T1906 BOOL  ; #1-1腔体氦检数据取值判定延时（测试）
T1907 BOOL  ; #1-1腔体抽残气压力到达延时（测试）
T1908 BOOL  ; #1-1腔体抽残气时间上限到达延时（测试）
T1909 BOOL  ; #1-1腔体预抽时间到达延时（测试）
T1910 BOOL  ; $?St$Bk?_#[195] / #1-1腔体真空在可氦检状态（测试） / $?St$Bk?_#[195]
T1920 BOOL  ; #1-1电池抽真空阈值到达延时（测试）
T1921 BOOL  ; #1-1电池抽真空时间上限到达延时（测试）
T1922 BOOL  ; #1-1电池破真空阈值到达延时（测试）
T1923 BOOL  ; #1-1电池破真空时间上限到达延时（测试）
T1924 BOOL  ; #1-1电池注氦压力到达延时（测试）
T1925 BOOL  ; #1-1电池注氦时间上限到达延时（测试）
T1926 BOOL  ; #1-1电池抽残气压力到达延时（测试）
T1927 BOOL  ; #1-1电池抽残气时间上限到达延时（测试）
T1928 BOOL  ; #1-1电池预抽压力正常判定延时（测试）
T1940 BOOL  ; 数据初始化延时（清氦）
T1941 BOOL  ; 清氦注氮时长（清氦）
T1980 BOOL  ; #1-1腔体数据初始化延时（标漏）
T1981 BOOL  ; #1-1腔体抽真空阀值到达延时（标漏）
T1982 BOOL  ; #1-1腔体抽真空时间上限到达延时（标漏）
T1984 BOOL  ; #1-1腔体氦检延时（标漏）
T1985 BOOL  ; #1-1腔体氦检数据取值完成判定（标漏）
T1986 BOOL  ; 氦检阀打开后，腔体压力超过氦检安全阀值，判氦检异常（标漏）
T1987 BOOL  ; 开氦检阀前抽气阀关延时（标漏）
T1990 BOOL  ; 氦检仪稳定延时（公共）
T2000 BOOL  ; #2-1腔体抽真空阈值到达延时（测试）
T2001 BOOL  ; #2-1腔体抽真空时间上限到达延时（测试）
T2002 BOOL  ; #2-1腔体破真空阈值到达延时（测试）
T2004 BOOL  ; #2-1腔体氦检时间（测试）
T2005 BOOL  ; #2-1腔体抽气阀关闭延时（测试）
T2006 BOOL  ; #2-1腔体氦检数据取值判定延时（测试）
T2007 BOOL  ; #2-1腔体抽残气压力到达延时（测试）
T2008 BOOL  ; #2-1腔体抽残气时间上限到达延时（测试）
T2009 BOOL  ; #2-1腔体预抽时间到达延时（测试）
T2010 BOOL  ; #2-1腔体真空在可氦检状态（测试）
T2020 BOOL  ; #2-1电池抽真空阈值到达延时（测试）
T2021 BOOL  ; #2-1电池抽真空时间上限到达延时（测试）
T2022 BOOL  ; #2-1电池破真空阈值到达延时（测试）
T2023 BOOL  ; #2-1电池破真空时间上限到达延时（测试）
T2024 BOOL  ; #2-1电池注氦压力到达延时（测试）
T2025 BOOL  ; #2-1电池注氦时间上限到达延时（测试）
T2026 BOOL  ; #2-1电池抽残气压力到达延时（测试）
T2027 BOOL  ; #2-1电池抽残气时间上限到达延时（测试）
T2028 BOOL  ; #2-1电池预抽压力正常判定延时（测试）
T2040 BOOL  ; #2-1数据初始化延时（清氦）
T2041 BOOL  ; #2-1清氦注氮时长（清氦）
T2081 BOOL  ; #2-1腔体抽真空阀值到达延时（标漏）
T2082 BOOL  ; #2-1腔体抽真空时间上限到达延时（标漏）
T2084 BOOL  ; #2-1腔体氦检延时（标漏）
T2085 BOOL  ; #2-1腔体氦检数据取值完成判定（标漏）
T2086 BOOL  ; #2-1氦检阀打开后，腔体压力超过氦检安全阀值，判氦检异常（标漏）
T2087 BOOL  ; #2-1开氦检阀前抽气阀关延时（标漏）
T2100 BOOL  ; #3-1腔体抽真空阈值到达延时（测试）
T2101 BOOL  ; #3-1腔体抽真空时间上限到达延时（测试）
T2102 BOOL  ; #3-1腔体破真空阈值到达延时（测试）
T2104 BOOL  ; #3-1腔体氦检时间（测试）
T2105 BOOL  ; #3-1腔体抽气阀关闭延时（测试）
T2106 BOOL  ; #3-1腔体氦检数据取值判定延时（测试）
T2107 BOOL  ; #3-1腔体抽残气压力到达延时（测试）
T2108 BOOL  ; #3-1腔体抽残气时间上限到达延时（测试）
T2109 BOOL  ; #3-1腔体预抽时间到达延时（测试）
T2110 BOOL  ; #3-1腔体真空在可氦检状态（测试）
T2120 BOOL  ; #3-1电池抽真空阈值到达延时（测试）
T2121 BOOL  ; #3-1电池抽真空时间上限到达延时（测试）
T2122 BOOL  ; #3-1电池破真空阈值到达延时（测试）
T2123 BOOL  ; #3-1电池破真空时间上限到达延时（测试）
T2124 BOOL  ; #3-1电池注氦压力到达延时（测试）
T2125 BOOL  ; #3-1电池注氦时间上限到达延时（测试）
T2126 BOOL  ; #3-1电池抽残气压力到达延时（测试）
T2127 BOOL  ; #3-1电池抽残气时间上限到达延时（测试）
T2128 BOOL  ; #3-1电池预抽压力正常判定延时（测试）
T2140 BOOL  ; #3-1数据初始化延时（清氦）
T2141 BOOL  ; #3-1清氦注氮时长（清氦）
T2181 BOOL  ; #3-1腔体抽真空阀值到达延时（标漏）
T2182 BOOL  ; #3-1腔体抽真空时间上限到达延时（标漏）
T2184 BOOL  ; #3-1腔体氦检延时（标漏）
T2185 BOOL  ; #3-1腔体氦检数据取值完成判定（标漏）
T2186 BOOL  ; #3-1氦检阀打开后，腔体压力超过氦检安全阀值，判氦检异常（标漏）
T2187 BOOL  ; #3-1开氦检阀前抽气阀关延时（标漏）
T2220 BOOL  ; #1-2电池抽真空阈值到达延时（测试）
T2221 BOOL  ; #1-2电池抽真空时间上限到达延时（测试）
T2222 BOOL  ; #1-2电池破真空阈值到达延时（测试）
T2223 BOOL  ; #1-2电池破真空时间上限到达延时（测试）
T2224 BOOL  ; #1-2电池注氦压力到达延时（测试）
T2225 BOOL  ; #1-2电池注氦时间上限到达延时（测试）
T2226 BOOL  ; #1-2电池抽残气压力到达延时（测试）
T2227 BOOL  ; #1-2电池抽残气时间上限到达延时（测试）
T2228 BOOL  ; #1-2电池预抽压力正常判定延时（测试）
T2281 BOOL  ; #1-2腔体抽真空阀值到达延时（标漏）
T2282 BOOL  ; #1-2腔体抽真空时间上限到达延时（标漏）
T2284 BOOL  ; #1-2腔体氦检延时（标漏）
T2286 BOOL  ; #1-2氦检阀打开后，腔体压力超过氦检安全阀值，判氦检异常（标漏）
T2287 BOOL  ; #1-2开氦检阀前抽气阀关延时（标漏）
T2320 BOOL  ; #2-2电池抽真空阈值到达延时（测试）
T2321 BOOL  ; #2-2电池抽真空时间上限到达延时（测试）
T2322 BOOL  ; #2-2电池破真空阈值到达延时（测试）
T2323 BOOL  ; #2-2电池破真空时间上限到达延时（测试）
T2324 BOOL  ; #2-2电池注氦压力到达延时（测试）
T2325 BOOL  ; #2-2电池注氦时间上限到达延时（测试）
T2326 BOOL  ; #2-2电池抽残气压力到达延时（测试）
T2327 BOOL  ; #2-2电池抽残气时间上限到达延时（测试）
T2328 BOOL  ; #2-2电池预抽压力正常判定延时（测试）
T2381 BOOL  ; #2-2腔体抽真空阀值到达延时（标漏）
T2382 BOOL  ; #2-2腔体抽真空时间上限到达延时（标漏）
T2384 BOOL  ; #2-2腔体氦检延时（标漏）
T2386 BOOL  ; #2-2氦检阀打开后，腔体压力超过氦检安全阀值，判氦检异常（标漏）
T2387 BOOL  ; #2-2开氦检阀前抽气阀关延时（标漏）
T2420 BOOL  ; #3-2电池抽真空阈值到达延时（测试）
T2421 BOOL  ; #3-2电池抽真空时间上限到达延时（测试）
T2422 BOOL  ; #3-2电池破真空阈值到达延时（测试）
T2423 BOOL  ; #3-2电池破真空时间上限到达延时（测试）
T2424 BOOL  ; #3-2电池注氦压力到达延时（测试）
T2425 BOOL  ; #3-2电池注氦时间上限到达延时（测试）
T2426 BOOL  ; #3-2电池抽残气压力到达延时（测试）
T2427 BOOL  ; #3-2电池抽残气时间上限到达延时（测试）
T2428 BOOL  ; #3-2电池预抽压力正常判定延时（测试）
T2481 BOOL  ; #3-2腔体抽真空阀值到达延时（标漏）
T2482 BOOL  ; #3-2腔体抽真空时间上限到达延时（标漏）
T2484 BOOL  ; #3-2腔体氦检延时（标漏）
T2486 BOOL  ; #3-2氦检阀打开后，腔体压力超过氦检安全阀值，判氦检异常（标漏）
T2487 BOOL  ; #3-2开氦检阀前抽气阀关延时（标漏）
T2521 BOOL  ; 进料#1扫码延时
T2522 BOOL  ; 接收数据清零延时发送无协议通讯TXD
T2523 BOOL  ; 进料#1扫码结果判定延时
T2524 BOOL  ; 进料#1扫码发送超时
T2531 BOOL  ; 进料#2扫码延时
T2532 BOOL  ; 扫码长度判定延时
T2600 BOOL  ; #4-1腔体抽真空阈值到达延时（测试）
T2601 BOOL  ; #4-1腔体抽真空时间上限到达延时（测试）
T2602 BOOL  ; #4-1腔体破真空阈值到达延时（测试）
T2603 BOOL  ; #4-1腔体破真空时间上限到达延时（测试）
T2604 BOOL  ; #4-1腔体氦检时间（测试）
T2605 BOOL  ; #4-1腔体抽气阀关闭延时（测试）
T2606 BOOL  ; #4-1腔体氦检数据取值判定延时（测试）
T2607 BOOL  ; #4-1腔体抽残气压力到达延时（测试）
T2608 BOOL  ; #4-1腔体抽残气时间上限到达延时（测试）
T2609 BOOL  ; #4-1腔体预抽时间到达延时（测试）
T2610 BOOL  ; #4-1腔体真空在可氦检状态（测试）
T2611 BOOL  ; #4-1腔体氦检时压力过高判定延时（测试）
T2612 BOOL  ; #4-1（测试）
T2613 BOOL  ; #4-1（测试）
T2614 BOOL  ; #4-1（测试）
T2615 BOOL  ; #4-1（测试）
T2616 BOOL  ; #4-1（测试）
T2617 BOOL  ; #4-1（测试）
T2618 BOOL  ; #4-1（测试）
T2619 BOOL  ; #4-1（测试）
T2620 BOOL  ; #4-1电池抽真空阈值到达延时（测试）
T2621 BOOL  ; #4-1电池抽真空时间上限到达延时（测试）
T2622 BOOL  ; #4-1电池破真空阈值到达延时（测试）
T2623 BOOL  ; #4-1电池破真空时间上限到达延时（测试）
T2624 BOOL  ; #4-1电池注氦压力到达延时（测试）
T2625 BOOL  ; #4-1电池注氦时间上限到达延时（测试）
T2626 BOOL  ; #4-1电池抽残气压力到达延时（测试）
T2627 BOOL  ; #4-1电池抽残气时间上限到达延时（测试）
T2628 BOOL  ; #4-1电池预抽压力正常判定延时（测试）
T2629 BOOL  ; #4-1（测试）
T2630 BOOL  ; #4-1（测试）
T2631 BOOL  ; #4-1（测试）
T2632 BOOL  ; #4-1（测试）
T2633 BOOL  ; #4-1（测试）
T2634 BOOL  ; #4-1（测试）
T2635 BOOL  ; #4-1（测试）
T2636 BOOL  ; #4-1（测试）
T2637 BOOL  ; #4-1（测试）
T2638 BOOL  ; #4-1（测试）
T2639 BOOL  ; #4-1（测试）
T2640 BOOL  ; #4-1数据初始化延时（清氦）
T2641 BOOL  ; #4-1清氦注氮时长（清氦）
T2642 BOOL  ; #4-1（测试）
T2643 BOOL  ; #4-1（测试）
T2644 BOOL  ; #4-1（测试）
T2645 BOOL  ; #4-1（测试）
T2646 BOOL  ; #4-1（测试）
T2647 BOOL  ; #4-1（测试）
T2648 BOOL  ; #4-1（测试）
T2649 BOOL  ; #4-1（测试）
T2680 BOOL  ; #4-1腔体数据初始化延时（标漏）
T2681 BOOL  ; #4-1腔体抽真空阀值到达延时（标漏）
T2682 BOOL  ; #4-1腔体抽真空时间上限到达延时（标漏）
T2683 BOOL  ; #4-1腔体真空值在可氦检状态（标漏）
T2684 BOOL  ; #4-1腔体氦检延时（标漏）
T2685 BOOL  ; #4-1腔体氦检数据取值完成判定（标漏）
T2686 BOOL  ; #4-1氦检阀打开后，腔体压力超过氦检安全阀值，判氦检异常（标漏）
T2687 BOOL  ; #4-1开氦检阀前抽气阀关延时（标漏）
T2700 BOOL  ; #4-2腔体抽真空阈值到达延时（测试）
T2701 BOOL  ; #4-2腔体抽真空时间上限到达延时（测试）
T2702 BOOL  ; #4-2腔体破真空阈值到达延时（测试）
T2703 BOOL  ; #4-2腔体破真空时间上限到达延时（测试）
T2704 BOOL  ; #4-2腔体氦检时间（测试）
T2705 BOOL  ; #4-2腔体抽气阀关闭延时（测试）
T2706 BOOL  ; #4-2腔体氦检数据取值判定延时（测试）
T2707 BOOL  ; #4-2腔体抽残气压力到达延时（测试）
T2708 BOOL  ; #4-2腔体抽残气时间上限到达延时（测试）
T2709 BOOL  ; #4-2腔体预抽时间到达延时（测试）
T2710 BOOL  ; #4-2腔体真空在可氦检状态（测试）
T2711 BOOL  ; #4-2腔体氦检时压力过高判定延时（测试）
T2712 BOOL  ; #4-2（测试）
T2713 BOOL  ; #4-2（测试）
T2714 BOOL  ; #4-2（测试）
T2715 BOOL  ; #4-2（测试）
T2716 BOOL  ; #4-2（测试）
T2717 BOOL  ; #4-2（测试）
T2718 BOOL  ; #4-2（测试）
T2719 BOOL  ; #4-2（测试）
T2720 BOOL  ; #4-2电池抽真空阈值到达延时（测试）
T2721 BOOL  ; #4-2电池抽真空时间上限到达延时（测试）
T2722 BOOL  ; #4-2电池破真空阈值到达延时（测试）
T2723 BOOL  ; #4-2电池破真空时间上限到达延时（测试）
T2724 BOOL  ; #4-2电池注氦压力到达延时（测试）
T2725 BOOL  ; #4-2电池注氦时间上限到达延时（测试）
T2726 BOOL  ; #4-2电池抽残气压力到达延时（测试）
T2727 BOOL  ; #4-2电池抽残气时间上限到达延时（测试）
T2728 BOOL  ; #4-2电池预抽压力正常判定延时（测试）
T2729 BOOL  ; #4-2（测试）
T2730 BOOL  ; #4-2（测试）
T2731 BOOL  ; #4-2（测试）
T2732 BOOL  ; #4-2（测试）
T2733 BOOL  ; #4-2（测试）
T2734 BOOL  ; #4-2（测试）
T2735 BOOL  ; #4-2（测试）
T2736 BOOL  ; #4-2（测试）
T2737 BOOL  ; #4-2（测试）
T2738 BOOL  ; #4-2（测试）
T2739 BOOL  ; #4-2（测试）
T2740 BOOL  ; #4-2数据初始化延时（清氦）
T2741 BOOL  ; #4-2清氦注氮时长（清氦）
T2742 BOOL  ; #4-2（测试）
T2743 BOOL  ; #4-2（测试）
T2744 BOOL  ; #4-2（测试）
T2745 BOOL  ; #4-2（测试）
T2746 BOOL  ; #4-2（测试）
T2747 BOOL  ; #4-2（测试）
T2748 BOOL  ; #4-2（测试）
T2749 BOOL  ; #4-2（测试）
T2780 BOOL  ; #4-2腔体数据初始化延时（标漏）
T2781 BOOL  ; #4-2腔体抽真空阀值到达延时（标漏）
T2782 BOOL  ; #4-2腔体抽真空时间上限到达延时（标漏）
T2783 BOOL  ; #4-2腔体真空值在可氦检状态（标漏）
T2784 BOOL  ; #4-2腔体氦检延时（标漏）
T2785 BOOL  ; #4-2腔体氦检数据取值完成判定（标漏）
T2786 BOOL  ; #4-2氦检阀打开后，腔体压力超过氦检安全阀值，判氦检异常（标漏）
T2787 BOOL  ; #4-2开氦检阀前抽气阀关延时（标漏）
T2800 BOOL  ; 复测腔体抽真空阈值到达延时（测试）
T2801 BOOL  ; 复测腔体抽真空时间上限到达延时（测试）
T2802 BOOL  ; 复测腔体破真空阈值到达延时（测试）
T2804 BOOL  ; 复测腔体氦检时间（测试）
T2805 BOOL  ; 复测腔体抽气阀关闭延时（测试）
T2806 BOOL  ; 复测腔体氦检数据取值判定延时（测试）
T2807 BOOL  ; 复测腔体抽残气压力到达延时（测试）
T2808 BOOL  ; 复测腔体抽残气时间上限到达延时（测试）
T2809 BOOL  ; 复测腔体预抽时间到达延时（测试）
T2810 BOOL  ; 复测腔体真空在可氦检状态（测试）
T2820 BOOL  ; 复测电池抽真空阈值到达延时（测试）
T2821 BOOL  ; 复测电池抽真空时间上限到达延时（测试）
T2822 BOOL  ; 复测电池破真空阈值到达延时（测试）
T2823 BOOL  ; 复测电池破真空时间上限到达延时（测试）
T2824 BOOL  ; 复测电池注氦压力到达延时（测试）
T2825 BOOL  ; 复测电池注氦时间上限到达延时（测试）
T2826 BOOL  ; 复测电池抽残气压力到达延时（测试）
T2827 BOOL  ; 复测电池抽残气时间上限到达延时（测试）
T2828 BOOL  ; 复测电池预抽压力正常判定延时（测试）
T2840 BOOL  ; 复测数据初始化延时（清氦）
T2841 BOOL  ; 复测清氦注氮时长（清氦）
T2849 BOOL  ; 复测开破真空阀延时（测试）
T3006 BOOL  ; #4腔体破真空阀开到位报警延时
T3007 BOOL  ; #4腔体破真空阀关到位报警延时
T3018 BOOL  ; #4-1电池破真空阀开到位报警延时
T3019 BOOL  ; #4-1电池破真空阀关到位报警延时
T3020 BOOL  ; #4-2电池破真空阀开到位报警延时
T3021 BOOL  ; #4-2电池破真空阀关到位报警延时
W0.00 BOOL  ; 启动按钮（SW）
W0.01 BOOL  ; 停止按钮(SW)
W0.02 BOOL  ; 复位按钮（SW）
W0.04 BOOL  ; 整机复位按钮（SW）
W0.05 BOOL  ; 清料停止按钮（SW）
W0.06 BOOL  ; 整机记忆清除（SW）
W0.07 BOOL  ; 门磁屏蔽（SW）
W0.08 BOOL  ; 蜂鸣器屏蔽（SW）
W0.14 BOOL  ; 进料拉带#1扫码测试[SW]
W0.15 BOOL  ; 进料拉带#2扫码测试[SW]
W100.00 BOOL  ; 扫码NG料满位标志
W100.01 BOOL  ; 氦检NG料满标志
W1.00 BOOL  ; 手动模式
W1.01 BOOL  ; 自动模式
W1.09 BOOL  ; 伺服进料允许（允许=0）
W1.10 BOOL  ; 上料位有料模拟
W1.11 BOOL  ; 清料时单个料有效选择
W1.15 BOOL  ; 有料记忆异常屏蔽（手动调试）
W200.00 BOOL  ; 进料拉带机构隔离位&扫码位&进料位全有料标志
W200.01 BOOL  ; 调试1
W200.02 BOOL  ; 调试2
W200.03 BOOL  ; 调试3
W204.00 BOOL  ; 来料拉带机构单步标志
W20.00 BOOL  ; 腔体真空泵M1停机1分钟内禁止启动保护
W20.01 BOOL  ; 氦检前置泵停机1分钟内禁止启动保护
W20.02 BOOL  ; 腔体真空泵M2停机1分钟内禁止启动保护
W210.00 BOOL  ; 进料伺服有取料需求标志
W210.01 BOOL  ; 进料伺服有放扫码NG料需求标志
W210.02 BOOL  ; 进料伺服有配对取/放料需求标志
W210.03 BOOL  ; 进料伺服有腔体放料需求标志
W211.00 BOOL  ; 进料伺服有配对放料需求标志
W211.01 BOOL  ; 进料伺服有配对取料需求标志
W211.02 BOOL  ; #1氦检腔有放料需求标志
W211.03 BOOL  ; #2氦检腔有放料需求标志
W211.04 BOOL  ; #3氦检腔有放料需求标志
W211.05 BOOL  ; #4氦检腔有放料需求标志
W230.00 BOOL  ; 出料模组X轴初始化完成
W230.03 BOOL  ; 下料模组X/Z运行许可
W231.00 BOOL  ; 出料伺服Z轴到待机位
W231.01 BOOL  ; 出料伺服X轴到#1腔取料位
W231.02 BOOL  ; 出料伺服X轴到#2腔取料位
W231.03 BOOL  ; 出料伺服X轴到#3腔取料位
W231.04 BOOL  ; 出料伺服Z轴到#1腔取料位
W231.05 BOOL  ; 出料伺服Z轴到#2腔取料位
W231.06 BOOL  ; 出料伺服Z轴到#3腔取料位
W231.07 BOOL  ; $?St$Bk?_#[196] / 下料Z模组到待机位 / $?St$Bk?_#[196]
W231.08 BOOL  ; 下料X模组到OK下料位
W231.09 BOOL  ; 下料Z模组到OK下料位
W231.10 BOOL  ; 下料Z模组到待机位
W231.11 BOOL  ; 出料伺服X轴到#4腔取料位
W231.12 BOOL  ; 出料伺服Z轴到#4腔取料位
W232 CHANNEL  ; INI_PV字
W234.00 BOOL  ; 出料Z轴到待机位
W234.01 BOOL  ; 出料X到位置
W234.02 BOOL  ; 出料Z轴到2#爪放NG位置
W234.03 BOOL  ; 出料Z轴回待机位
W234.04 BOOL  ; 出料X到放NG（复测缓存）位置
W234.05 BOOL  ; 出料Z轴到放NG（复测缓存）位置
W234.06 BOOL  ; 出料Z轴回待机位
W236.00 BOOL  ; 出料Z模组到待机位
W236.01 BOOL  ; 出料伺服X轴到#2夹爪氦检NG放料位
W236.02 BOOL  ; 出料伺服X轴到#1夹爪氦检NG放料位
W236.03 BOOL  ; 出料伺服z轴到#2夹爪氦检NG放料位
W236.04 BOOL  ; 出料伺服Z轴到#1夹爪氦检NG放料位
W236.05 BOOL  ; 出料Z轴到待机位
W236.06 BOOL  ; 出料伺服X轴到缓存配对取料位
W236.07 BOOL  ; 出料伺服X轴到#位
W236.09 BOOL  ; 出料伺服Z轴到#1夹爪配对取放料位
W236.10 BOOL  ; 出料伺服Z轴到#2夹爪配对取放料位
W236.11 BOOL  ; 出料伺服Z轴到待机位
W236.12 BOOL  ; 出料伺服X轴到位
W236.13 BOOL  ; 出料伺服z轴到OK放料位
W236.14 BOOL  ; 出料Z轴到待机位
W240.00 BOOL  ; 出料模组Z轴初始化完成
W2.00 BOOL  ; 清料按钮（SW）
W2.01 BOOL  ; 设备PPM计数启动按钮（SW）
W30.00 BOOL  ; #1来料位有料标志
W30.01 BOOL  ; #1隔离位有料标志
W30.02 BOOL  ; #1扫码阻挡有料标志
W30.03 BOOL  ; #1进料位有料标志
W31.00 BOOL  ; #2来料位有料标志
W31.01 BOOL  ; #2隔离位有料标志
W31.02 BOOL  ; #2扫码阻挡有料标志
W31.03 BOOL  ; #2进料位有料标志
W360.03 BOOL  ; 进料伺服X轴取料位设定按钮(SW)
W360.04 BOOL  ; 进料伺服X轴#1腔放料位设定按钮(SW)
W360.05 BOOL  ; 进料伺服X轴#2腔放料位设定按钮(SW)
W360.06 BOOL  ; 进料伺服X轴#3腔放料位设定按钮(SW)
W360.07 BOOL  ; 进料伺服X轴#1夹爪扫码NG放料位设定按钮(SW)
W360.08 BOOL  ; 进料伺服X轴#2夹爪扫码NG放料位设定按钮(SW)
W360.09 BOOL  ; 进料伺服X轴#1夹爪配对取放料位设定按钮(SW)
W360.10 BOOL  ; 进料伺服X轴#2夹爪配对取放料位设定按钮(SW)
W360.11 BOOL  ; 进料伺服X轴#1腔有料检测位设定按钮(SW)
W360.12 BOOL  ; 进料伺服X轴#2腔有料检测位设定按钮(SW)
W360.13 BOOL  ; 进料伺服X轴#3腔有料检测位设定按钮(SW)
W360.14 BOOL  ; 进料伺服X轴#4腔放料位设定按钮(SW)
W361.03 BOOL  ; 进料伺服X轴取料位触发标志
W361.04 BOOL  ; 进料伺服X轴#1腔放料位触发标志
W361.05 BOOL  ; 进料伺服X轴#2腔放料位触发标志
W361.06 BOOL  ; 进料伺服X轴#3腔放料位触发标志
W361.07 BOOL  ; 进料伺服X轴#1夹爪扫码NG放料位触发标志
W361.08 BOOL  ; 进料伺服X轴#2夹爪扫码NG放料位触发标志
W361.09 BOOL  ; 进料伺服X轴#1夹爪配对取放料位触发标志
W361.10 BOOL  ; 进料伺服X轴#2夹爪配对取放料位触发标志
W361.11 BOOL  ; 进料伺服X轴#1腔有料检测位触发标志
W361.12 BOOL  ; 进料伺服X轴#2腔有料检测位触发标志
W361.13 BOOL  ; 进料伺服X轴#3腔有料检测位触发标志
W361.14 BOOL  ; 进料伺服X轴#4腔放料位触发标志
W362.03 BOOL  ; 进料伺服Z轴待机位设定按钮(SW)
W363.03 BOOL  ; 进料伺服Z轴待机位触发标志
W363.04 BOOL  ; 进料伺服Z轴取料位触发标志
W363.05 BOOL  ; 进料伺服Z轴#1腔放料位触发标志
W363.06 BOOL  ; 进料伺服Z轴#2腔放料位触发标志
W363.07 BOOL  ; 进料伺服Z轴#3腔放料位触发标志
W363.08 BOOL  ; 进料伺服Z轴#1夹爪扫码NG放料位触发标志
W363.09 BOOL  ; 进料伺服Z轴#2夹爪扫码NG放料位触发标志
W363.10 BOOL  ; 进料伺服Z轴#1夹爪配对取放料位触发标志
W363.11 BOOL  ; 进料伺服Z轴#2夹爪配对取放料位触发标志
W363.12 BOOL  ; 进料伺服Z轴#4腔放料位触发标志
W365.03 BOOL  ; 复测伺服X轴待机位设定按钮(SW)
W365.04 BOOL  ; 复测伺服X轴测试腔体位设定按钮(SW)
W365.05 BOOL  ; 复测伺服X轴#1取料位设定按钮(SW)
W365.06 BOOL  ; 复测伺服X轴#2取料位设定按钮(SW)
W365.07 BOOL  ; 复测伺服X轴#1配对位设定按钮(SW)
W365.08 BOOL  ; 复测伺服X轴#2配对位设定按钮(SW)
W365.09 BOOL  ; 复测伺服X轴NG放料位设定按钮(SW)
W366.03 BOOL  ; 复测伺服X轴待机位触发标志
W366.04 BOOL  ; 复测伺服X轴测试腔体位触发标志
W366.05 BOOL  ; 复测伺服X轴#1取料位触发标志
W366.06 BOOL  ; 复测伺服X轴#2取料位触发标志
W366.07 BOOL  ; 复测伺服X轴#1配对位触发标志
W366.08 BOOL  ; 复测伺服X轴#2配对位触发标志
W366.09 BOOL  ; 复测伺服X轴NG放料位触发标志
W367.03 BOOL  ; 复测伺服Z轴待机位设定按钮(SW)
W367.04 BOOL  ; 复测伺服Z轴取料位设定按钮(SW)
W367.05 BOOL  ; 复测伺服Z轴OK放料位设定按钮(SW)
W367.06 BOOL  ; 复测伺服Z轴NG放料位设定按钮(SW)
W367.07 BOOL  ; 复测伺服Z轴腔体取放料位设定按钮(SW)
W368.03 BOOL  ; 复测伺服Z轴待机位触发标志
W368.04 BOOL  ; 复测伺服Z轴取料位触发标志
W368.05 BOOL  ; 复测伺服Z轴OK放料位触发标志
W368.06 BOOL  ; 复测伺服Z轴NG放料位触发标志
W368.07 BOOL  ; 复测伺服Z轴腔体取放料位触发标志
W370.03 BOOL  ; 出料伺服X轴放料位设定按钮(SW)
W370.04 BOOL  ; 出料伺服X轴#1腔取料位设定按钮(SW)
W370.05 BOOL  ; 出料伺服X轴#2腔取料位设定按钮(SW)
W370.06 BOOL  ; 出料伺服X轴#3腔取料位设定按钮(SW)
W370.07 BOOL  ; 出料伺服X轴#1夹爪氦检NG放料位设定按钮(SW)
W370.08 BOOL  ; 出料伺服X轴#2夹爪氦检NG放料位设定按钮(SW)
W370.09 BOOL  ; 出料伺服X轴#1夹爪配对取放料位设定按钮(SW)
W370.10 BOOL  ; 出料伺服X轴#2夹爪配对取放料位设定按钮(SW)
W370.11 BOOL  ; 出料伺服X轴#4腔取料位设定按钮(SW)
W371.03 BOOL  ; 出料伺服X轴放料位触发标志
W371.04 BOOL  ; 出料伺服X轴#1腔取料位触发标志
W371.05 BOOL  ; 出料伺服X轴#2腔取料位触发标志
W371.06 BOOL  ; 出料伺服X轴#3腔取料位触发标志
W371.07 BOOL  ; 出料伺服X轴#1夹爪氦检NG放料位触发标志
W371.08 BOOL  ; 出料伺服X轴#2夹爪氦检NG放料位触发标志
W371.09 BOOL  ; 出料伺服X轴#1夹爪配对取放料位触发标志
W371.10 BOOL  ; 出料伺服X轴#2夹爪配对取放料位触发标志
W371.14 BOOL  ; 出料伺服X轴#4腔取料位触发标志
W372.03 BOOL  ; 出料伺服Z轴待机位设定按钮(SW)
W373.03 BOOL  ; 出料伺服Z轴待机位触发标志
W373.04 BOOL  ; 出料伺服Z轴放料位触发标志
W373.05 BOOL  ; 出料伺服Z轴#1腔取料位触发标志
W373.06 BOOL  ; 出料伺服Z轴#2腔取料位触发标志
W373.07 BOOL  ; 出料伺服Z轴#3腔取料位触发标志
W373.08 BOOL  ; 出料伺服Z轴#1夹爪氦检NG放料位触发标志
W373.09 BOOL  ; 出料伺服Z轴#2夹爪氦检NG放料位触发标志
W373.10 BOOL  ; 出料伺服Z轴#1夹爪配对取放料位触发标志
W373.11 BOOL  ; 出料伺服Z轴#2夹爪配对取放料位触发标志
W380.01 BOOL  ; 读氦检仪状态完成
W380.06 BOOL  ; 读氦检仪检漏口压力完成
W380.11 BOOL  ; 读氦检仪漏率完成
W380.15 BOOL  ; 氦检仪漏率低于设定值（稳态）
W381.00 BOOL  ; 氦检仪在检漏状态
W381.03 BOOL  ; 氦检仪在启动状态
W3.00 BOOL  ; 氦检单双检测选择允许
W400 CHANNEL  ; 设备故障
W400.00 BOOL  ; #1扫码阻挡气缸缩回位[alm]
W400.01 BOOL  ; #1扫码阻挡气缸伸出位[alm]
W400.02 BOOL  ; #1隔离气缸缩回位[alm]
W400.03 BOOL  ; #1隔离气缸伸出位[alm]
W400.04 BOOL  ; #2扫码阻挡气缸缩回位[alm]
W400.05 BOOL  ; #2扫码阻挡气缸伸出位[alm]
W400.06 BOOL  ; #2隔离气缸缩回位[alm]
W400.07 BOOL  ; #2隔离气缸伸出位 [alm]
W400.08 BOOL  ; #1进料夹爪夹紧位[alm]
W400.09 BOOL  ; #1进料夹爪松开位[alm]
W400.10 BOOL  ; #2进料夹爪夹紧位[alm]
W400.11 BOOL  ; #2进料夹爪松开位[alm]
W400.12 BOOL  ; 进料夹爪变距气缸伸出位[alm]
W400.13 BOOL  ; 进料夹爪变距气缸缩回位[alm]
W400.14 BOOL  ; #1出料夹爪夹紧位[alm]
W400.15 BOOL  ; #1出料夹爪松开位[alm]
W401.00 BOOL  ; #2出料夹爪夹紧位[alm]
W401.01 BOOL  ; #2出料夹爪松开位[alm]
W401.02 BOOL  ; 出料夹爪变距气缸伸出位[alm]
W401.03 BOOL  ; 出料夹爪变距气缸缩回位[alm]
W401.04 BOOL  ; #1腔体平移一级气缸缩回位[alm]
W401.05 BOOL  ; #1腔体平移一级气缸伸出位[alm]
W401.06 BOOL  ; #1腔体平移二级气缸缩回位[alm]
W401.07 BOOL  ; #1腔体平移二级气缸伸出位[alm]
W401.08 BOOL  ; #1腔体顶伸气缸上升位[alm]
W401.09 BOOL  ; #1腔体顶伸气缸下降位[alm]
W401.10 BOOL  ; #1腔体氦检阀开到位[alm]
W401.11 BOOL  ; #1腔体氦检阀关到位[alm]
W401.12 BOOL  ; #1腔体有料感应1[alm]
W401.13 BOOL  ; #1腔体有料感应2[alm]
W401.14 BOOL  ; 0[alm]
W401.15 BOOL  ; 0[alm]
W402.00 BOOL  ; 0[alm]
W402.01 BOOL  ; #2腔体平移一级气缸缩回位[alm]
W402.02 BOOL  ; #2腔体平移一级气缸伸出位[alm]
W402.03 BOOL  ; #2腔体平移二级气缸缩回位[alm]
W402.04 BOOL  ; #2腔体平移二级气缸伸出位[alm]
W402.05 BOOL  ; #2腔体顶伸气缸上升位[alm]
W402.06 BOOL  ; #2腔体顶伸气缸下降位[alm]
W402.07 BOOL  ; #2腔体氦检阀开到位[alm]
W402.08 BOOL  ; #2腔体氦检阀关到位[alm]
W402.09 BOOL  ; 2#腔体有料感应1[alm]
W402.10 BOOL  ; 2#腔体有料感应2[alm]
W402.11 BOOL  ; 0[alm]
W402.12 BOOL  ; 0[alm]
W402.13 BOOL  ; 0[alm]
W402.14 BOOL  ; #3腔体平移一级气缸缩回位[alm]
W402.15 BOOL  ; #3腔体平移一级气缸伸出位[alm]
W403.00 BOOL  ; #3腔体平移二级气缸缩回位[alm]
W403.01 BOOL  ; #3腔体平移二级气缸伸出位[alm]
W403.02 BOOL  ; #3腔体顶伸气缸上升位[alm]
W403.03 BOOL  ; #3腔体顶伸气缸下降位[alm]
W403.04 BOOL  ; #3腔体氦检阀开到位[alm]
W403.05 BOOL  ; #3腔体氦检阀关到位[alm]
W403.06 BOOL  ; 氦检仪准备好了信号[alm]
W403.07 BOOL  ; 氦检仪故障信号[alm]
W403.08 BOOL  ; #3腔体有料感应1[alm]
W403.09 BOOL  ; #3腔体有料感应2[alm]
W403.10 BOOL  ; 0[alm]
W403.11 BOOL  ; 进料伺服X轴准备好了信号[alm]
W403.12 BOOL  ; 进料伺服X轴故障信号[alm]
W403.13 BOOL  ; 进料伺服Z轴准备好了信号[alm]
W403.14 BOOL  ; 进料伺服Z轴故障信号[alm]
W403.15 BOOL  ; 0[alm]
W404.00 BOOL  ; 出料伺服X轴准备好了信号[alm]
W404.01 BOOL  ; 出料伺服X轴故障信号[alm]
W404.02 BOOL  ; 出料伺服Z轴准备好了信号[alm]
W404.03 BOOL  ; 出料伺服Z轴故障信号[alm]
W404.04 BOOL  ; 0[alm]
W404.05 BOOL  ; 腔体抽真空泵运行信号[alm]
W404.06 BOOL  ; 腔体抽真空泵过载信号[alm]
W404.07 BOOL  ; 氦检前置泵运行信号[alm]
W404.08 BOOL  ; 氦检前置泵过载信号[alm]
W404.09 BOOL  ; 启动按钮[alm]
W404.10 BOOL  ; 停止按钮[alm]
W404.11 BOOL  ; 复位按钮[alm]
W404.12 BOOL  ; 急停按钮[alm]
W404.13 BOOL  ; 手自动选择[alm]
W404.14 BOOL  ; #1进料夹爪防下坠感应[alm]
W404.15 BOOL  ; #2进料夹爪防下坠感应[alm]
W405.00 BOOL  ; #1出料夹爪防下坠感应[alm]
W405.01 BOOL  ; #2出料夹爪防下坠感应[alm]
W405.02 BOOL  ; 0[alm]
W405.03 BOOL  ; 进料对接输入[alm]
W405.04 BOOL  ; 出料对接输入[alm]
W405.05 BOOL  ; 0[alm]
W405.06 BOOL  ; 0[alm]
W405.07 BOOL  ; 设备总气压信号[alm]
W405.08 BOOL  ; #1来料位有料感应[alm]
W405.09 BOOL  ; #2来料位有料感应[alm]
W405.10 BOOL  ; #1隔离位有料感应[alm]
W405.11 BOOL  ; #2隔离位有料感应[alm]
W405.12 BOOL  ; #1扫码位有料感应[alm]
W405.13 BOOL  ; #2扫码位有料感应[alm]
W405.14 BOOL  ; #1-1进料位有料感应[alm]
W405.15 BOOL  ; #1-2进料位有料感应[alm]
W406.00 BOOL  ; #2-1进料位有料感应[alm]
W406.01 BOOL  ; #2-2进料位有料感应[alm]
W406.02 BOOL  ; 进料夹爪柔性感应[alm]
W406.03 BOOL  ; 出料夹爪柔性感应[alm]
W406.04 BOOL  ; #1进料夹爪对应腔体有料感应[alm]
W406.05 BOOL  ; #2进料夹爪对应腔体有料感应[alm]
W406.06 BOOL  ; 扫码NG放料#1位有料感应[alm]
W406.07 BOOL  ; 扫码NG放料#2位有料感应[alm]
W406.08 BOOL  ; 扫码NG料满位有料感应[alm]
W406.09 BOOL  ; 进料配对位有料感应[alm]
W406.10 BOOL  ; 出料配对位有料感应[alm]
W406.11 BOOL  ; 氦检NG放料#1位有料感应[alm]
W406.12 BOOL  ; 氦检NG放料#2位有料感应[alm]
W406.13 BOOL  ; 氦检NG料满位有料感应[alm]
W406.14 BOOL  ; #1-1出料位有料感应[alm]
W406.15 BOOL  ; #1-2出料位有料感应[alm]
W407.00 BOOL  ; #2-1出料位有料感应[alm]
W407.01 BOOL  ; #2-2出料位有料感应[alm]
W407.02 BOOL  ; #1门磁开关[alm]
W407.03 BOOL  ; #2门磁开关[alm]
W407.04 BOOL  ; #3门磁开关[alm]
W407.05 BOOL  ; #4门磁开关[alm]
W407.06 BOOL  ; #5门磁开关[alm]
W407.07 BOOL  ; #6门磁开关[alm]
W407.08 BOOL  ; #7门磁开关[alm]
W407.09 BOOL  ; #8门磁开关[alm]
W407.10 BOOL  ; #9门磁开关[alm]
W407.11 BOOL  ; #10门磁开关[alm]
W407.12 BOOL  ; #11门磁开关[alm]
W407.13 BOOL  ; #12门磁开关[alm]
W407.14 BOOL  ; #13门磁开关[alm]
W407.15 BOOL  ; #14门磁开关[alm]
W411.00 BOOL  ; 电脑软件未启动[alm]
W411.01 BOOL  ; 氦检仪通信异常[alm]
W411.02 BOOL  ; #1扫码枪通讯异常[alm]
W411.03 BOOL  ; #2扫码枪通讯异常[alm]
W411.04 BOOL  ; 进料扫码MES入站就绪通知&确认超时[alm]
W411.05 BOOL  ; 出料伺服MES出站就绪通知&确认超时[alm]
W413.00 BOOL  ; 进料伺服X轴正极限[alm]
W413.01 BOOL  ; 进料伺服X轴负极限[alm]
W413.02 BOOL  ; 进料伺服X轴原点[alm]
W413.03 BOOL  ; 进料伺服Z轴正极限[alm]
W413.04 BOOL  ; 进料伺服Z轴负极限[alm]
W413.05 BOOL  ; 进料伺服Z轴原点[alm]
W413.06 BOOL  ; 出料伺服X轴正极限[alm]
W413.07 BOOL  ; 出料伺服X轴负极限[alm]
W413.08 BOOL  ; 出料伺服X轴原点[alm]
W413.09 BOOL  ; 出料伺服Z轴正极限[alm]
W413.10 BOOL  ; 出料伺服Z轴负极限[alm]
W413.11 BOOL  ; 出料伺服Z轴原点[alm]
W414.00 BOOL  ; 氦检仪不在检漏状态[alm]
W414.14 BOOL  ; 整机复位超时[alm]
W414.15 BOOL  ; 进料拉带工站复位超时[alm]
W415.00 BOOL  ; 进料伺服工站复位超时[alm]
W415.01 BOOL  ; #1氦检工站复位超时[alm]
W415.02 BOOL  ; #2氦检工站复位超时[alm]
W415.03 BOOL  ; #3氦检工站复位超时[alm]
W415.04 BOOL  ; 出料伺服工站复位超时[alm]
W415.05 BOOL  ; $?St$Bk?_#[197] / #4氦检工站复位超时[alm] / $?St$Bk?_#[197]
W415.10 BOOL  ; 氦检仪未启动，请检查
W415.11 BOOL  ; 进料拉带连续入栈#1次数超过3次
W415.12 BOOL  ; 进料拉带连续入栈#2次数超过3次
W415.13 BOOL  ; 电池抽残气超过2次
W416.00 BOOL  ; #1来料位有料记忆[alm]
W416.01 BOOL  ; #2来料位有料记忆[alm]
W416.02 BOOL  ; #1隔离位有料记忆[alm]
W416.03 BOOL  ; #2隔离位有料记忆[alm]
W416.04 BOOL  ; #1扫码位有料记忆[alm]
W416.05 BOOL  ; #2扫码位有料记忆[alm]
W416.06 BOOL  ; #1进料位有料记忆[alm]
W416.07 BOOL  ; #2进料位有料记忆[alm]
W416.08 BOOL  ; #1进料夹爪有料记忆[alm]
W416.09 BOOL  ; #2进料夹爪有料记忆[alm]
W416.10 BOOL  ; #1出料夹爪有料记忆[alm]
W416.11 BOOL  ; #2出料夹爪有料记忆[alm]
W416.12 BOOL  ; #1-1腔体有料记忆[alm]
W416.13 BOOL  ; #1-2腔体有料记忆[alm]
W416.14 BOOL  ; #2-1腔体有料记忆[alm]
W416.15 BOOL  ; #2-2腔体有料记忆[alm]
W417.00 BOOL  ; #3-1腔体有料记忆[alm]
W417.01 BOOL  ; #3-2腔体有料记忆[alm]
W417.02 BOOL  ; 进料配对位有料记忆[alm]
W417.03 BOOL  ; 出料配对位有料记忆[alm]
W417.04 BOOL  ; #1出料位有料记忆[alm]
W417.05 BOOL  ; #2出料位有料记忆[alm]
W417.06 BOOL  ; 扫码NG放料位有料记忆[alm]
W417.07 BOOL  ; 氦检NG拉带下料位有料记忆[alm]
W418.00 BOOL  ; 整机复位超时[alm]
W418.01 BOOL  ; 进料拉带工站复位超时[alm]
W418.02 BOOL  ; 进料伺服工站复位超时[alm]
W418.03 BOOL  ; #1氦检工站复位超时[alm]
W418.04 BOOL  ; #2氦检工站复位超时[alm]
W418.05 BOOL  ; #3氦检工站复位超时[alm]
W418.06 BOOL  ; 出料伺服工站复位超时[alm]
W418.07 BOOL  ; #4氦检工站复位超时[alm]
W418.08 BOOL  ; 复测移载机构工站复位超时
W418.09 BOOL  ; 复测腔体机构工站复位超时
W420.14 BOOL  ; #1腔体抽真空阀开到位[alm]
W420.15 BOOL  ; #1腔体抽真空阀关到位[alm]
W421.00 BOOL  ; #1-1腔体阀开到位[alm]
W421.01 BOOL  ; #1-1腔体阀关到位[alm]
W421.02 BOOL  ; #1-2腔体阀开到位[alm]
W421.03 BOOL  ; #1-2腔体阀关到位[alm]
W421.04 BOOL  ; #1腔体破真空阀开到位[alm]
W421.05 BOOL  ; #1腔体破真空阀关到位[alm]
W421.06 BOOL  ; #1腔体顶部吹气开到位[alm]
W421.07 BOOL  ; #1腔体顶部吹气关到位[alm]
W421.08 BOOL  ; #2腔体抽真空阀开到位[alm]
W421.09 BOOL  ; #2腔体抽真空阀关到位[alm]
W421.10 BOOL  ; #2-1腔体阀开到位[alm]
W421.11 BOOL  ; #2-1腔体阀关到位[alm]
W421.12 BOOL  ; #2-2腔体阀开到位[alm]
W421.13 BOOL  ; #2-2腔体阀关到位[alm]
W421.14 BOOL  ; #2腔体破真空阀开到位[alm]
W421.15 BOOL  ; #2腔体破真空阀关到位[alm]
W422.00 BOOL  ; #2腔体顶部吹气开到位[alm]
W422.01 BOOL  ; #2腔体顶部吹气关到位[alm]
W422.02 BOOL  ; #3腔体抽真空阀开到位[alm]
W422.03 BOOL  ; #3腔体抽真空阀关到位[alm]
W422.04 BOOL  ; #3-1腔体阀开到位[alm]
W422.05 BOOL  ; #3-1腔体阀关到位[alm]
W422.06 BOOL  ; #3-2腔体阀开到位[alm]
W422.07 BOOL  ; #3-2腔体阀关到位[alm]
W422.08 BOOL  ; #3腔体破真空阀开到位[alm]
W422.09 BOOL  ; #3腔体破真空阀关到位[alm]
W422.10 BOOL  ; #3腔体顶部吹气开到位[alm]
W422.11 BOOL  ; #3腔体顶部吹气关到位[alm]
W422.12 BOOL  ; #1-1电池抽真空阀开到位[alm]
W422.13 BOOL  ; #1-1电池抽真空阀关到位[alm]
W422.14 BOOL  ; #1-2电池抽真空阀开到位[alm]
W422.15 BOOL  ; #1-2电池抽真空阀关到位[alm]
W423.00 BOOL  ; #1-1电池注氦阀开到位[alm]
W423.01 BOOL  ; #1-1电池注氦阀关到位[alm]
W423.02 BOOL  ; #1-2电池注氦阀开到位[alm]
W423.03 BOOL  ; #1-2电池注氦阀关到位[alm]
W423.04 BOOL  ; #1-1电池破真空阀开到位[alm]
W423.05 BOOL  ; #1-1电池破真空阀关到位[alm]
W423.06 BOOL  ; #1-2电池破真空阀开到位[alm]
W423.07 BOOL  ; #1-2电池破真空阀关到位[alm]
W423.08 BOOL  ; #2-1电池抽真空阀开到位[alm]
W423.09 BOOL  ; #2-1电池抽真空阀关到位[alm]
W423.10 BOOL  ; #2-2电池抽真空阀开到位[alm]
W423.11 BOOL  ; #2-2电池抽真空阀关到位[alm]
W423.12 BOOL  ; #2-1电池注氦阀开到位[alm]
W423.13 BOOL  ; #2-1电池注氦阀关到位[alm]
W423.14 BOOL  ; #2-2电池注氦阀开到位[alm]
W423.15 BOOL  ; #2-2电池注氦阀关到位[alm]
W424.00 BOOL  ; #2-1电池破真空阀开到位[alm]
W424.01 BOOL  ; #2-1电池破真空阀关到位[alm]
W424.02 BOOL  ; #2-2电池破真空阀开到位[alm]
W424.03 BOOL  ; #2-2电池破真空阀关到位[alm]
W424.04 BOOL  ; #3-1电池抽真空阀开到位[alm]
W424.05 BOOL  ; #3-1电池抽真空阀关到位[alm]
W424.06 BOOL  ; #3-2电池抽真空阀开到位[alm]
W424.07 BOOL  ; #3-2电池抽真空阀关到位[alm]
W424.08 BOOL  ; #3-1电池注氦阀开到位[alm]
W424.09 BOOL  ; #3-1电池注氦阀关到位[alm]
W424.10 BOOL  ; #3-2电池注氦阀开到位[alm]
W424.11 BOOL  ; #3-2电池注氦阀关到位[alm]
W424.12 BOOL  ; #3-1电池破真空阀开到位[alm]
W424.13 BOOL  ; #3-1电池破真空阀关到位[alm]
W424.14 BOOL  ; #3-2电池破真空阀开到位[alm]
W424.15 BOOL  ; #3-2电池破真空阀关到位[alm]
W425.00 BOOL  ; #4腔体抽真空阀开到位[alm]
W425.01 BOOL  ; #4腔体抽真空阀关到位[alm]
W425.02 BOOL  ; #4-1腔体阀开到位[alm]
W425.03 BOOL  ; #4-1腔体阀关到位[alm]
W425.04 BOOL  ; #4-2腔体阀开到位[alm]
W425.05 BOOL  ; #4-2腔体阀关到位[alm]
W425.06 BOOL  ; #4腔体破真空阀开到位[alm]
W425.07 BOOL  ; #4腔体破真空阀关到位[alm]
W425.08 BOOL  ; #4腔体顶部吹气开到位[alm]
W425.09 BOOL  ; #4腔体顶部吹气关到位[alm]
W425.10 BOOL  ; #4-1电池抽真空阀开到位[alm]
W425.11 BOOL  ; #4-1电池抽真空阀关到位[alm]
W425.12 BOOL  ; #4-2电池抽真空阀开到位[alm]
W425.13 BOOL  ; #4-2电池抽真空阀关到位[alm]
W425.14 BOOL  ; #4-1电池注氦阀开到位[alm]
W425.15 BOOL  ; #4-1电池注氦阀关到位[alm]
W426.00 BOOL  ; #4-2电池注氦阀开到位[alm]
W426.01 BOOL  ; #4-2电池注氦阀关到位[alm]
W426.02 BOOL  ; #4-1电池破真空阀开到位[alm]
W426.03 BOOL  ; #4-1电池破真空阀关到位[alm]
W426.04 BOOL  ; #4-2电池破真空阀开到位[alm]
W426.05 BOOL  ; #4-2电池破真空阀关到位[alm]
W430.00 BOOL  ; #15门磁开关[alm]
W430.01 BOOL  ; #16门磁开关[alm]
W430.02 BOOL  ; #进料位对射光电有料感应[alm]
W430.03 BOOL  ; 0[alm]
W430.04 BOOL  ; #4腔体平移一级气缸缩回位[alm]
W430.05 BOOL  ; #4腔体平移一级气缸伸出位[alm]
W430.06 BOOL  ; #4腔体平移二级气缸缩回位[alm]
W430.07 BOOL  ; #4腔体平移二级气缸伸出位[alm]
W430.08 BOOL  ; #4腔体顶伸气缸上升位[alm]
W430.09 BOOL  ; #4腔体顶伸气缸下降位[alm]
W430.10 BOOL  ; #4腔体氦检阀开到位[alm]
W430.11 BOOL  ; #4腔体氦检阀关到位[alm]
W430.12 BOOL  ; 4#腔体有料感应1[alm]
W430.13 BOOL  ; 4#腔体有料感应2[alm]
W430.14 BOOL  ; 0[alm]
W430.15 BOOL  ; 0[alm]
W431.00 BOOL  ; 复测夹爪气缸夹紧位[alm]
W431.01 BOOL  ; 复测夹爪气缸松开位[alm]
W431.02 BOOL  ; 复检夹爪柔性感应[alm]
W431.03 BOOL  ; 复测腔体移栽气缸缩回位[alm]
W431.04 BOOL  ; 复测腔体移栽气缸伸出位[alm]
W431.05 BOOL  ; 复测腔体顶升气缸缩回位[alm]
W431.06 BOOL  ; 复测腔体顶升气缸伸出位[alm]
W431.07 BOOL  ; 复测腔体氦检阀开到位[alm]
W431.08 BOOL  ; 复测腔体氦检阀关到位[alm]
W431.09 BOOL  ; 复测腔体感应有料感应[alm]
W431.10 BOOL  ; 0[alm]
W431.11 BOOL  ; 出料配对位有料感应2[alm]
W431.12 BOOL  ; 0[alm]
W431.13 BOOL  ; 0[alm]
W431.14 BOOL  ; 0[alm]
W431.15 BOOL  ; 0[alm]
W432.00 BOOL  ; 腔体抽真空泵M2运行信号[alm]
W432.01 BOOL  ; 腔体抽真空泵M2过载信号[alm]
W432.02 BOOL  ; 测伺服X轴准备好信号[alm]
W432.03 BOOL  ; 复测伺服X轴故障信号[alm]
W432.04 BOOL  ; 复测伺服Z轴准备好信号[alm]
W432.05 BOOL  ; 复测伺服Z轴故障信号[alm]
W432.06 BOOL  ; 0[alm]
W432.07 BOOL  ; 0[alm]
W432.08 BOOL  ; 0[alm]
W432.09 BOOL  ; 0[alm]
W432.10 BOOL  ; 设备真空压力信号#1[alm]
W432.11 BOOL  ; 设备真空压力信号#2[alm]
W432.12 BOOL  ; 设备氦气压力信号#1[alm]
W432.13 BOOL  ; 设备氦气压力信号#2[alm]
W432.14 BOOL  ; 设备注氦压力调节阀#1[alm]
W432.15 BOOL  ; 设备注氦压力调节阀#2[alm]
W433.00 BOOL  ; 复测缓存拨料气缸缩回位[alm]
W433.01 BOOL  ; 复测缓存拨料气缸伸出位[alm]
W433.02 BOOL  ; 复测缓存顶升气缸缩回位[alm]
W433.03 BOOL  ; 复测缓存顶升气缸伸出位[alm]
W433.04 BOOL  ; 复测缓存#1有料感应1[alm]
W433.05 BOOL  ; 复测缓存#1有料感应2[alm]
W433.06 BOOL  ; 复测缓存#1有料感应3[alm]
W433.07 BOOL  ; 复测缓存#1有料感应4[alm]
W433.08 BOOL  ; 复测缓存#2有料感应1[alm]
W433.09 BOOL  ; 复测缓存#2有料感应2[alm]
W433.10 BOOL  ; 复测缓存#2有料感应3[alm]
W433.11 BOOL  ; 复测缓存#2有料感应4[alm]
W433.12 BOOL  ; 0[alm]
W433.13 BOOL  ; 0[alm]
W433.14 BOOL  ; 0[alm]
W433.15 BOOL  ; 0[alm]
W434.00 BOOL  ; #4腔体抽真空阀开到位[alm]
W434.01 BOOL  ; #4腔体抽真空阀关到位[alm]
W434.02 BOOL  ; #4-1腔体阀开到位[alm]
W434.03 BOOL  ; #4-1腔体阀关到位[alm]
W434.04 BOOL  ; #4-2腔体阀开到位[alm]
W434.05 BOOL  ; #4-2腔体阀关到位[alm]
W434.06 BOOL  ; #4腔体破真空阀开到位[alm]
W434.07 BOOL  ; #4腔体破真空阀关到位[alm]
W434.08 BOOL  ; #4腔体吹气阀开到位[alm]
W434.09 BOOL  ; #4腔体吹气阀关到位[alm]
W434.10 BOOL  ; #4-1电池抽真空阀开到位[alm]
W434.11 BOOL  ; #4-1电池抽真空阀关到位[alm]
W434.12 BOOL  ; #4-2电池抽真空阀开到位[alm]
W434.13 BOOL  ; #4-2电池抽真空阀关到位[alm]
W434.14 BOOL  ; #4-1电池注氦阀开到位[alm]
W434.15 BOOL  ; #4-1电池注氦阀关到位[alm]
W435.00 BOOL  ; #4-2电池注氦阀开到位[alm]
W435.01 BOOL  ; #4-2电池注氦阀关到位[alm]
W435.02 BOOL  ; #4-1电池破真空阀开到位[alm]
W435.03 BOOL  ; #4-1电池破真空阀关到位[alm]
W435.04 BOOL  ; #4-2电池破真空阀开到位[alm]
W435.05 BOOL  ; #4-2电池破真空阀关到位[alm]
W435.10 BOOL  ; [W435.10）复测腔体破真空异常,请检查[0000.10]
W436.02 BOOL  ; 复测电池破真空[alm]
W436.04 BOOL  ; [W436.04]复测夹爪有料记忆异常,请检查[0000.04]
W437.00 BOOL  ; 1#腔体模拟量断线检测
W437.01 BOOL  ; 2#腔体模拟量断线检测
W437.02 BOOL  ; 3#腔体模拟量断线检测
W437.03 BOOL  ; 4#腔体模拟量断线检测
W437.04 BOOL  ; 5#腔体模拟量断线检测
W437.06 BOOL  ; 5#电池模拟量断线检测
W437.08 BOOL  ; 1-1电池模拟量断线检测
W437.09 BOOL  ; 1-2电池模拟量断线检测
W437.10 BOOL  ; 2-1电池模拟量断线检测
W437.11 BOOL  ; 2-2电池模拟量断线检测
W437.12 BOOL  ; 3-1电池模拟量断线检测
W437.13 BOOL  ; 3-2电池模拟量断线检测
W437.14 BOOL  ; 4-1电池模拟量断线检测
W437.15 BOOL  ; 4-2电池模拟量断线检测
W4.00 BOOL  ; 初次上电#1腔体平移一级气缸伸出条件
W4.01 BOOL  ; 初次上电#1腔体平移二级气缸伸出条件
W4.02 BOOL  ; 初次上电#2腔体平移一级气缸伸出条件
W4.03 BOOL  ; 初次上电#2腔体平移二级气缸伸出条件
W4.04 BOOL  ; 初次上电#3腔体平移一级气缸伸出条件
W4.05 BOOL  ; 初次上电#3腔体平移二级气缸伸出条件
W4.06 BOOL  ; 初次上电#4腔体平移一级气缸伸出条件
W4.07 BOOL  ; 初次上电#4腔体平移二级气缸伸出条件
W5.05 BOOL  ; #1扫码料到位
W5.06 BOOL  ; #2扫码料到位
W65.00 BOOL  ; 进料#1扫码
W65.01 BOOL  ; 进料#1扫码发送
W65.02 BOOL  ; 进料#1扫码失败
W65.03 BOOL  ; 进料#1扫码成功
W65.04 BOOL  ; 进料#1扫码接收
W65.05 BOOL  ; 进料扫码重新触发
W6.00 BOOL  ; 1腔体NG次数过多
W6.01 BOOL  ; 2腔体NG次数过多
W6.02 BOOL  ; 3腔体NG次数过多
W6.03 BOOL  ; 4腔体NG次数过多
W75.00 BOOL  ; 进料#2扫码
W75.01 BOOL  ; 进料#2扫码发送
W75.02 BOOL  ; 进料#2扫码失败
W75.03 BOOL  ; 进料#2扫码成功
W75.04 BOOL  ; 进料#2扫码接收
W75.05 BOOL  ; 进料#2扫码重新触发
Battery_Vaccum_1_1 SMC混压表
Battery_Vaccum_1_2 SMC混压表
Battery_Vaccum_2_1 SMC混压表
Battery_Vaccum_2_2 SMC混压表
Battery_Vaccum_3_1 SMC混压表
Battery_Vaccum_3_2 SMC混压表
HJY 氦检仪
Vaccum_1 真空计
Vaccum_2 真空计
Vaccum_3 真空计
二号腔体自检 腔体自检
复测腔 SMC混压表
复检腔 真空计
复检腔体自检 腔体自检
三号腔体自检 腔体自检
四号腔体自检 腔体自检
一号腔体自检 腔体自检

## Program Main (cyclic task 0)
Local symbols
D CHANNEL  ; 进料#1扫码数据开始字

### Section Main

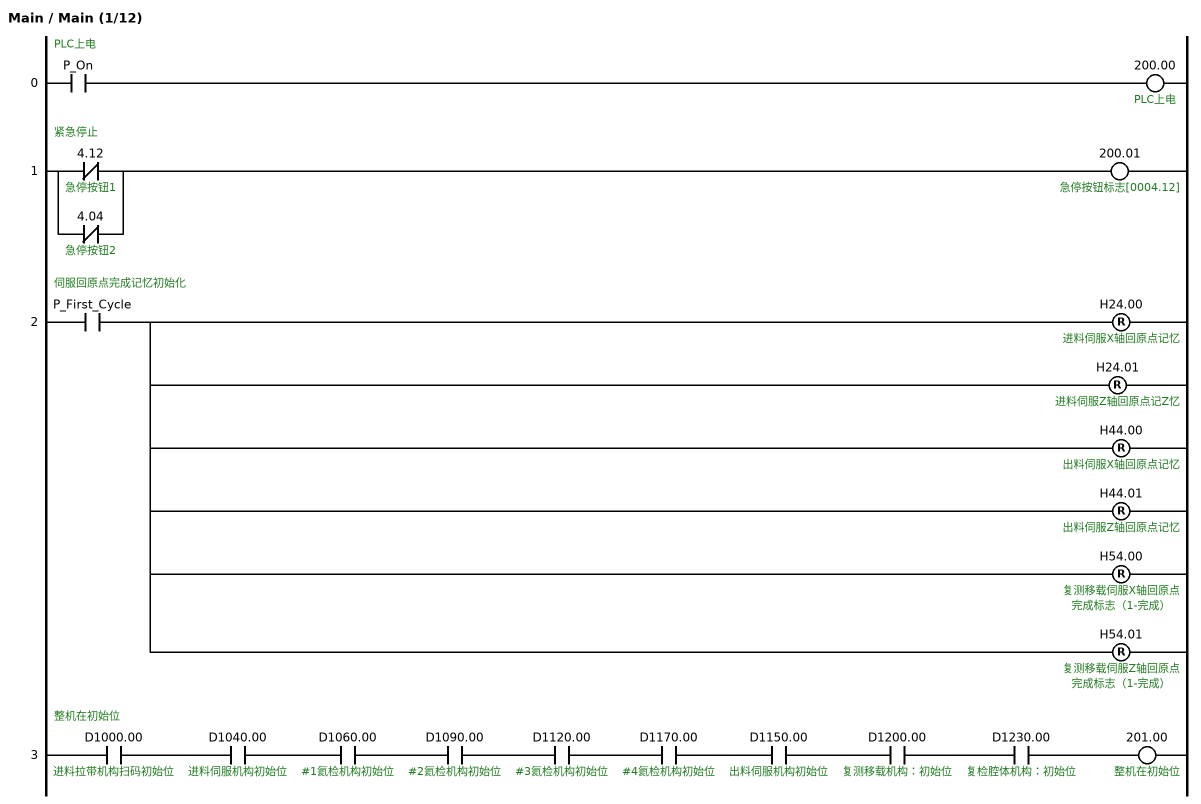
; rung 0: PLC上电
LD P_On
OUT 200.00  ; PLC上电
; rung 1: 紧急停止
LDNOT 4.12  ; 急停按钮1
ORNOT 4.04  ; 急停按钮2
OUT 200.01  ; 急停按钮标志[0004.12]
; rung 2: 伺服回原点完成记忆初始化
LD P_First_Cycle
RSET H24.00  ; 进料伺服X轴回原点记忆
RSET H24.01  ; 进料伺服Z轴回原点记Z忆
RSET H44.00  ; 出料伺服X轴回原点记忆
RSET H44.01  ; 出料伺服Z轴回原点记忆
RSET H54.00  ; 复测移载伺服X轴回原点完成标志（1-完成）
RSET H54.01  ; 复测移载伺服Z轴回原点完成标志（1-完成）
; rung 3: 整机在初始位
LD D1000.00  ; 进料拉带机构扫码初始位
AND D1040.00  ; 进料伺服机构初始位
AND D1060.00  ; #1氦检机构初始位
AND D1090.00  ; #2氦检机构初始位
AND D1120.00  ; #3氦检机构初始位
AND D1170.00  ; #4氦检机构初始位
AND D1150.00  ; 出料伺服机构初始位
AND D1200.00  ; 复测移载机构：初始位
AND D1230.00  ; 复检腔体机构：初始位
OUT 201.00  ; 整机在初始位

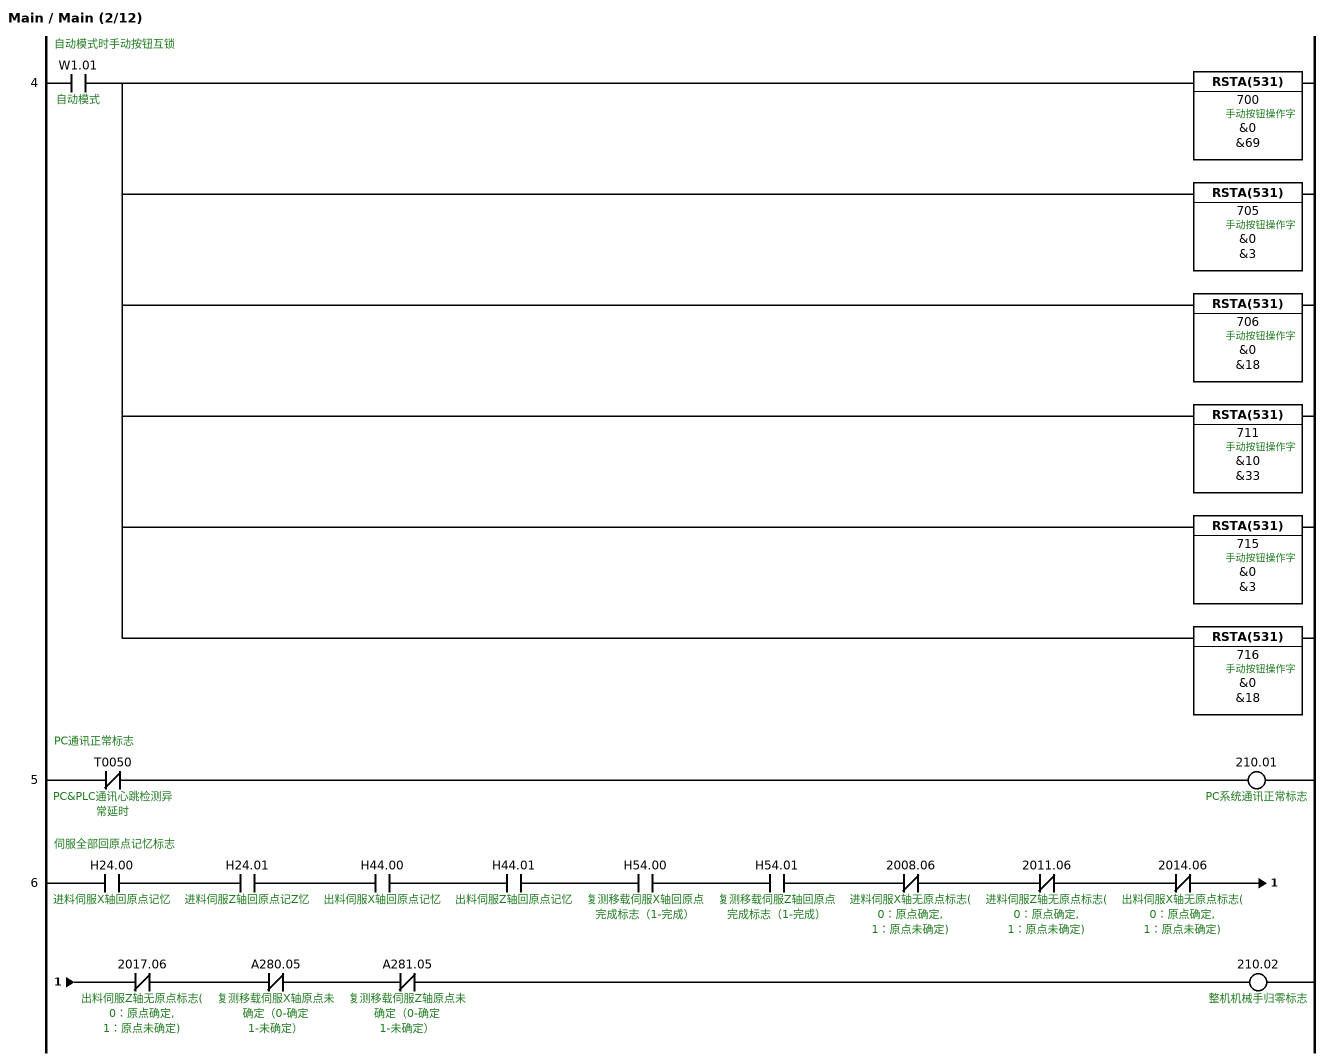
; rung 4: 自动模式时手动按钮互锁
LD W1.01  ; 自动模式
RSTA(531) 700 &0 &69  ; 手动按钮操作字
RSTA(531) 705 &0 &3  ; 手动按钮操作字
RSTA(531) 706 &0 &18  ; 手动按钮操作字
RSTA(531) 711 &10 &33  ; 手动按钮操作字
RSTA(531) 715 &0 &3  ; 手动按钮操作字
RSTA(531) 716 &0 &18  ; 手动按钮操作字
; rung 5: PC通讯正常标志
LDNOT T0050  ; PC&PLC通讯心跳检测异常延时
OUT 210.01  ; PC系统通讯正常标志
; rung 6: 伺服全部回原点记忆标志
LD H24.00  ; 进料伺服X轴回原点记忆
AND H24.01  ; 进料伺服Z轴回原点记Z忆
AND H44.00  ; 出料伺服X轴回原点记忆
AND H44.01  ; 出料伺服Z轴回原点记忆
AND H54.00  ; 复测移载伺服X轴回原点完成标志（1-完成）
AND H54.01  ; 复测移载伺服Z轴回原点完成标志（1-完成）
ANDNOT 2008.06  ; 进料伺服X轴无原点标志(0：原点确定,1：原点未确定)
ANDNOT 2011.06  ; 进料伺服Z轴无原点标志(0：原点确定,1：原点未确定)
ANDNOT 2014.06  ; 出料伺服X轴无原点标志(0：原点确定,1：原点未确定)
ANDNOT 2017.06  ; 出料伺服Z轴无原点标志(0：原点确定,1：原点未确定)
ANDNOT A280.05  ; 复测移载伺服X轴原点未确定（0-确定  1-未确定）
ANDNOT A281.05  ; 复测移载伺服Z轴原点未确定（0-确定  1-未确定）
OUT 210.02  ; 整机机械手归零标志

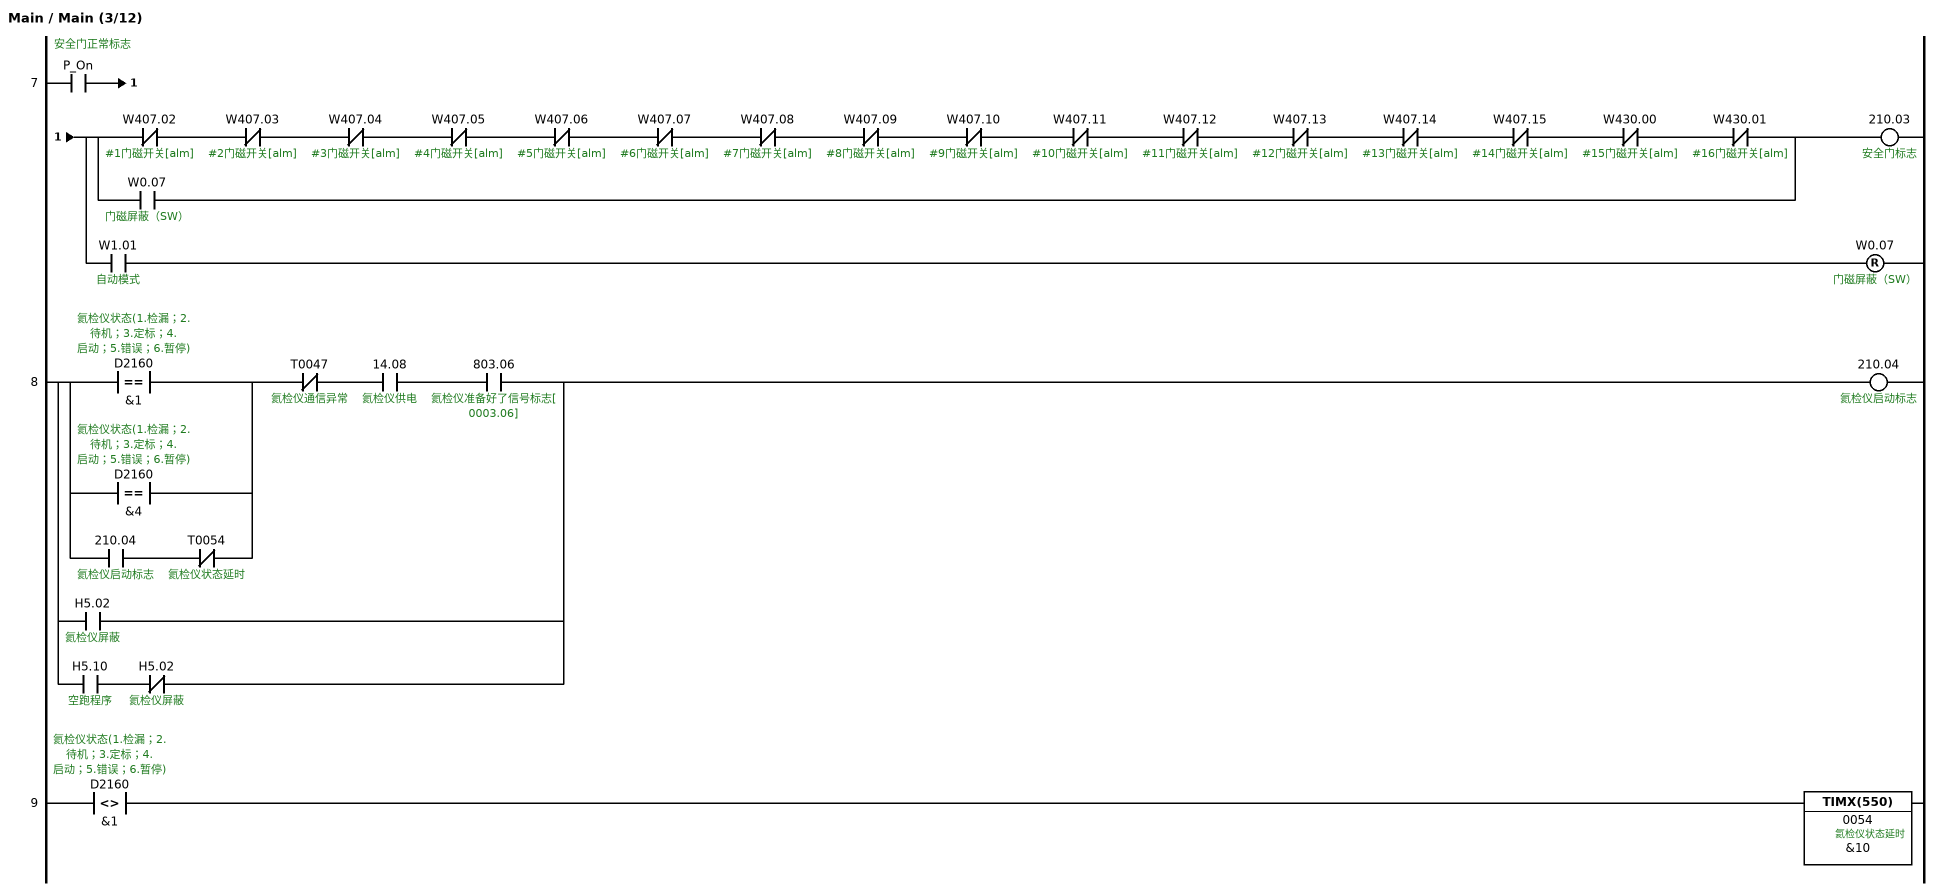
; rung 7: 安全门正常标志
LD P_On
OUT TR0
LDNOT W407.02  ; #1门磁开关[alm]
ANDNOT W407.03  ; #2门磁开关[alm]
ANDNOT W407.04  ; #3门磁开关[alm]
ANDNOT W407.05  ; #4门磁开关[alm]
ANDNOT W407.06  ; #5门磁开关[alm]
ANDNOT W407.07  ; #6门磁开关[alm]
ANDNOT W407.08  ; #7门磁开关[alm]
ANDNOT W407.09  ; #8门磁开关[alm]
ANDNOT W407.10  ; #9门磁开关[alm]
ANDNOT W407.11  ; #10门磁开关[alm]
ANDNOT W407.12  ; #11门磁开关[alm]
ANDNOT W407.13  ; #12门磁开关[alm]
ANDNOT W407.14  ; #13门磁开关[alm]
ANDNOT W407.15  ; #14门磁开关[alm]
ANDNOT W430.00  ; #15门磁开关[alm]
ANDNOT W430.01  ; #16门磁开关[alm]
OR W0.07  ; 门磁屏蔽（SW）
ANDLD
OUT 210.03  ; 安全门标志
LD TR0
AND W1.01  ; 自动模式
RSET W0.07  ; 门磁屏蔽（SW）
; rung 8
LD=(300) D2160 &1  ; 氦检仪状态(1.检漏；2.待机；3.定标；4.启动；5.错误；6.暂停)
OR=(300) D2160 &4  ; 氦检仪状态(1.检漏；2.待机；3.定标；4.启动；5.错误；6.暂停)
LD 210.04  ; 氦检仪启动标志
ANDNOT T0054  ; 氦检仪状态延时
ORLD
ANDNOT T0047  ; 氦检仪通信异常
AND 14.08  ; 氦检仪供电
AND 803.06  ; 氦检仪准备好了信号标志[0003.06]
OR H5.02  ; 氦检仪屏蔽
LD H5.10  ; 空跑程序
ANDNOT H5.02  ; 氦检仪屏蔽
ORLD
OUT 210.04  ; 氦检仪启动标志
; rung 9
LD<>(305) D2160 &1  ; 氦检仪状态(1.检漏；2.待机；3.定标；4.启动；5.错误；6.暂停)
TIMX(550) 0054 &10  ; 氦检仪状态延时

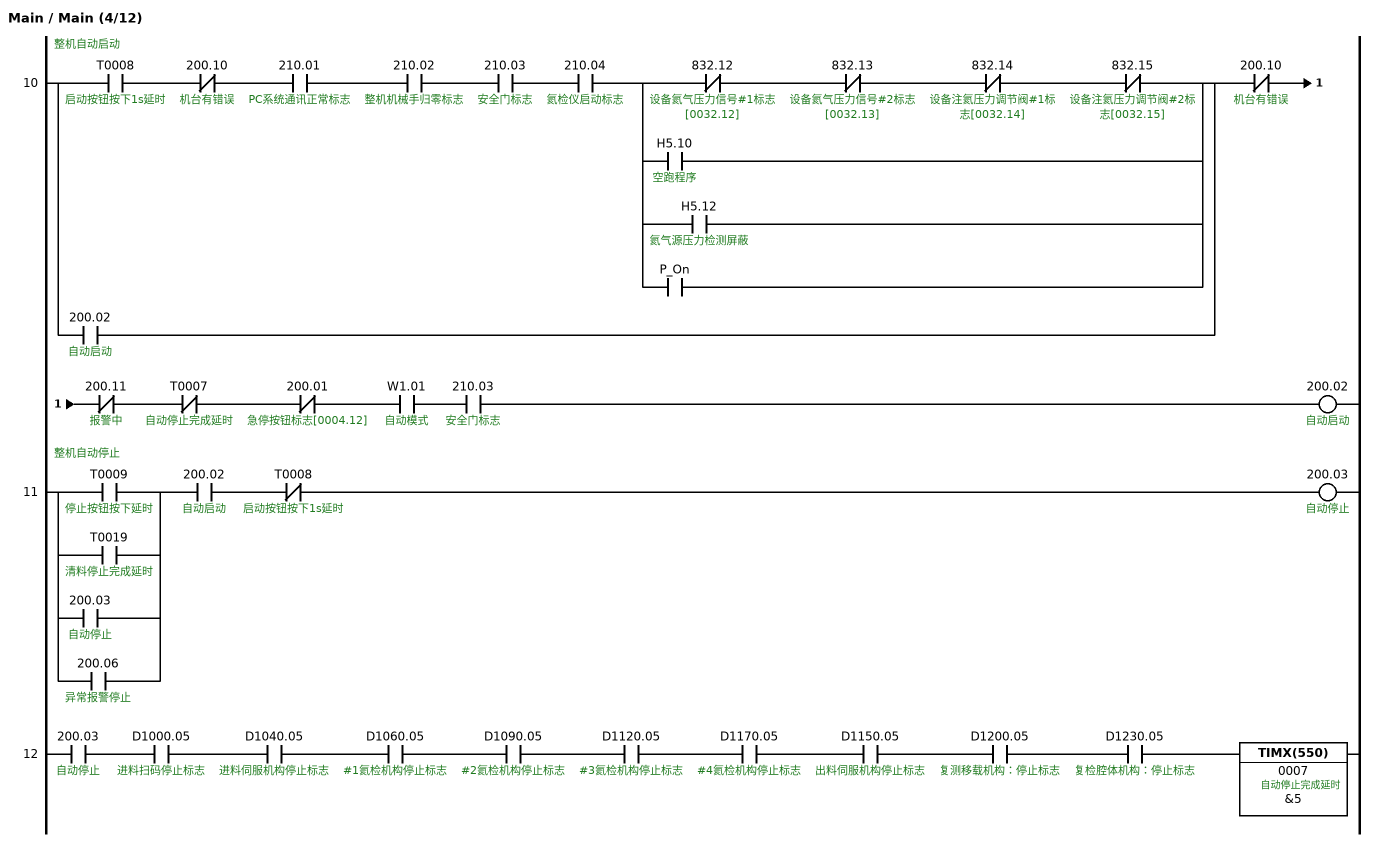
; rung 10: 整机自动启动
LD T0008  ; 启动按钮按下1s延时
ANDNOT 200.10  ; 机台有错误
AND 210.01  ; PC系统通讯正常标志
AND 210.02  ; 整机机械手归零标志
AND 210.03  ; 安全门标志
AND 210.04  ; 氦检仪启动标志
LDNOT 832.12  ; 设备氦气压力信号#1标志[0032.12]
ANDNOT 832.13  ; 设备氦气压力信号#2标志[0032.13]
ANDNOT 832.14  ; 设备注氦压力调节阀#1标志[0032.14]
ANDNOT 832.15  ; 设备注氦压力调节阀#2标志[0032.15]
OR H5.10  ; 空跑程序
OR H5.12  ; 氦气源压力检测屏蔽
OR P_On
ANDLD
OR 200.02  ; 自动启动
ANDNOT 200.10  ; 机台有错误
ANDNOT 200.11  ; 报警中
ANDNOT T0007  ; 自动停止完成延时
ANDNOT 200.01  ; 急停按钮标志[0004.12]
AND W1.01  ; 自动模式
AND 210.03  ; 安全门标志
OUT 200.02  ; 自动启动
; rung 11: 整机自动停止
LD T0009  ; 停止按钮按下延时
OR T0019  ; 清料停止完成延时
OR 200.03  ; 自动停止
OR 200.06  ; 异常报警停止
AND 200.02  ; 自动启动
ANDNOT T0008  ; 启动按钮按下1s延时
OUT 200.03  ; 自动停止
; rung 12
LD 200.03  ; 自动停止
AND D1000.05  ; 进料扫码停止标志
AND D1040.05  ; 进料伺服机构停止标志
AND D1060.05  ; #1氦检机构停止标志
AND D1090.05  ; #2氦检机构停止标志
AND D1120.05  ; #3氦检机构停止标志
AND D1170.05  ; #4氦检机构停止标志
AND D1150.05  ; 出料伺服机构停止标志
AND D1200.05  ; 复测移载机构：停止标志
AND D1230.05  ; 复检腔体机构：停止标志
TIMX(550) 0007 &5  ; 自动停止完成延时

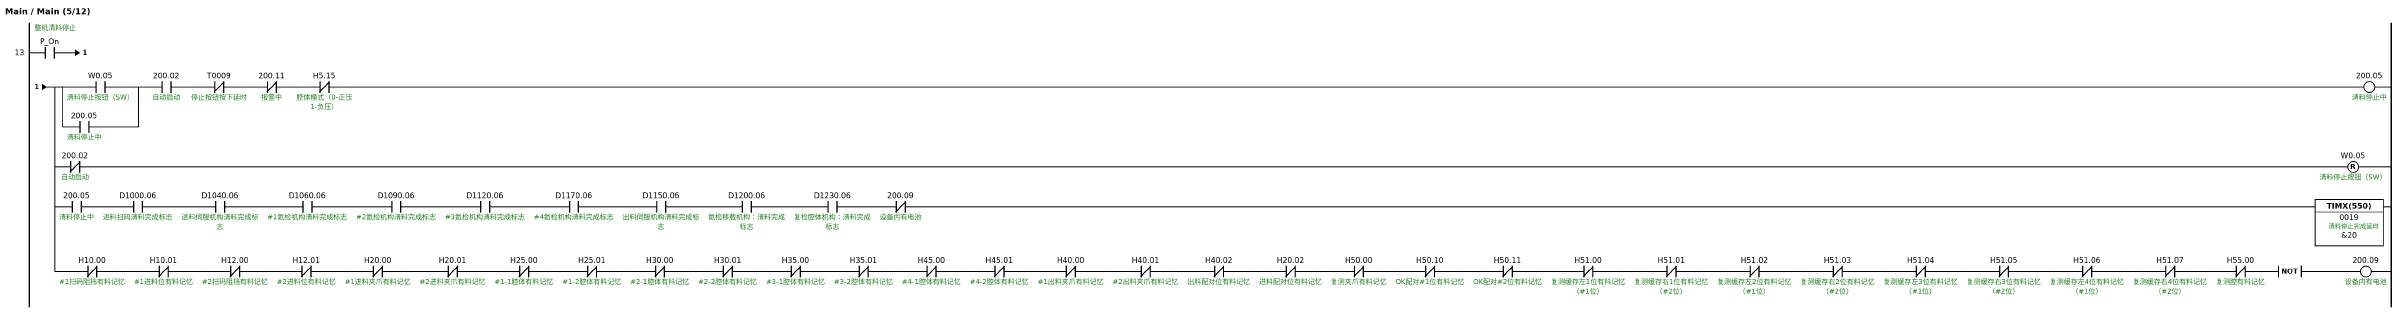
; rung 13: 整机清料停止
LD P_On
OUT TR0
LD W0.05  ; 清料停止按钮（SW）
OR 200.05  ; 清料停止中
ANDLD
AND 200.02  ; 自动启动
ANDNOT T0009  ; 停止按钮按下延时
ANDNOT 200.11  ; 报警中
ANDNOT H5.15  ; 腔体模式（0-正压 1-负压）
OUT 200.05  ; 清料停止中
LD TR0
ANDNOT 200.02  ; 自动启动
RSET W0.05  ; 清料停止按钮（SW）
LD TR0
AND 200.05  ; 清料停止中
AND D1000.06  ; 进料扫码清料完成标志
AND D1040.06  ; 进料伺服机构清料完成标志
AND D1060.06  ; #1氦检机构清料完成标志
AND D1090.06  ; #2氦检机构清料完成标志
AND D1120.06  ; #3氦检机构清料完成标志
AND D1170.06  ; #4氦检机构清料完成标志
AND D1150.06  ; 出料伺服机构清料完成标志
AND D1200.06  ; 氦检移载机构：清料完成标志
AND D1230.06  ; 复检腔体机构：清料完成标志
ANDNOT 200.09  ; 设备内有电池
TIMX(550) 0019 &20  ; 清料停止完成延时
LD TR0
ANDNOT H10.00  ; #1扫码阻挡有料记忆
ANDNOT H10.01  ; #1进料位有料记忆
ANDNOT H12.00  ; #2扫码阻挡有料记忆
ANDNOT H12.01  ; #2进料位有料记忆
ANDNOT H20.00  ; #1进料夹爪有料记忆
ANDNOT H20.01  ; #2进料夹爪有料记忆
ANDNOT H25.00  ; #1-1腔体有料记忆
ANDNOT H25.01  ; #1-2腔体有料记忆
ANDNOT H30.00  ; #2-1腔体有料记忆
ANDNOT H30.01  ; #2-2腔体有料记忆
ANDNOT H35.00  ; #3-1腔体有料记忆
ANDNOT H35.01  ; #3-2腔体有料记忆
ANDNOT H45.00  ; #4-1腔体有料记忆
ANDNOT H45.01  ; #4-2腔体有料记忆
ANDNOT H40.00  ; #1出料夹爪有料记忆
ANDNOT H40.01  ; #2出料夹爪有料记忆
ANDNOT H40.02  ; 出料配对位有料记忆
ANDNOT H20.02  ; 进料配对位有料记忆
ANDNOT H50.00  ; 复测夹爪有料记忆
ANDNOT H50.10  ; OK配对#1位有料记忆
ANDNOT H50.11  ; OK配对#2位有料记忆
ANDNOT H51.00  ; 复测缓存左1位有料记忆（#1位）
ANDNOT H51.01  ; 复测缓存右1位有料记忆（#2位）
ANDNOT H51.02  ; 复测缓存左2位有料记忆（#1位）
ANDNOT H51.03  ; 复测缓存右2位有料记忆（#2位）
ANDNOT H51.04  ; 复测缓存左3位有料记忆（#1位）
ANDNOT H51.05  ; 复测缓存右3位有料记忆（#2位）
ANDNOT H51.06  ; 复测缓存左4位有料记忆（#1位）
ANDNOT H51.07  ; 复测缓存右4位有料记忆（#2位）
ANDNOT H55.00  ; 复测腔有料记忆
NOT(520)
OUT 200.09  ; 设备内有电池

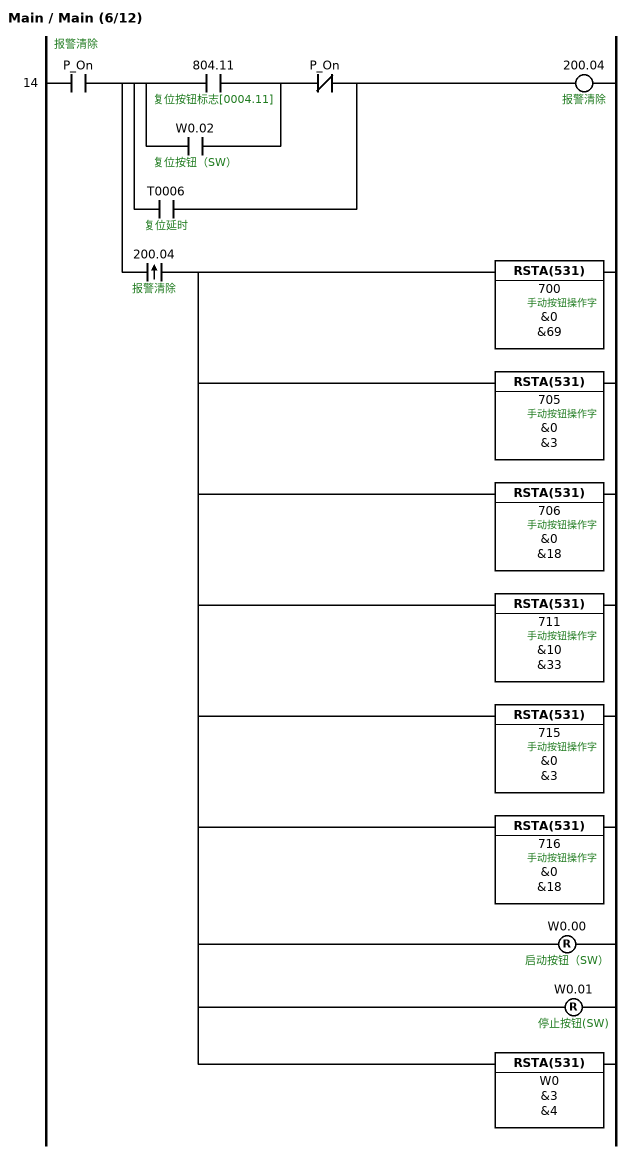
; rung 14: 报警清除
LD P_On
OUT TR0
LD 804.11  ; 复位按钮标志[0004.11]
OR W0.02  ; 复位按钮（SW）
ANDNOT P_On
OR T0006  ; 复位延时
ANDLD
OUT 200.04  ; 报警清除
LD TR0
@AND 200.04  ; 报警清除
RSTA(531) 700 &0 &69  ; 手动按钮操作字
RSTA(531) 705 &0 &3  ; 手动按钮操作字
RSTA(531) 706 &0 &18  ; 手动按钮操作字
RSTA(531) 711 &10 &33  ; 手动按钮操作字
RSTA(531) 715 &0 &3  ; 手动按钮操作字
RSTA(531) 716 &0 &18  ; 手动按钮操作字
RSET W0.00  ; 启动按钮（SW）
RSET W0.01  ; 停止按钮(SW)
RSTA(531) W0 &3 &4

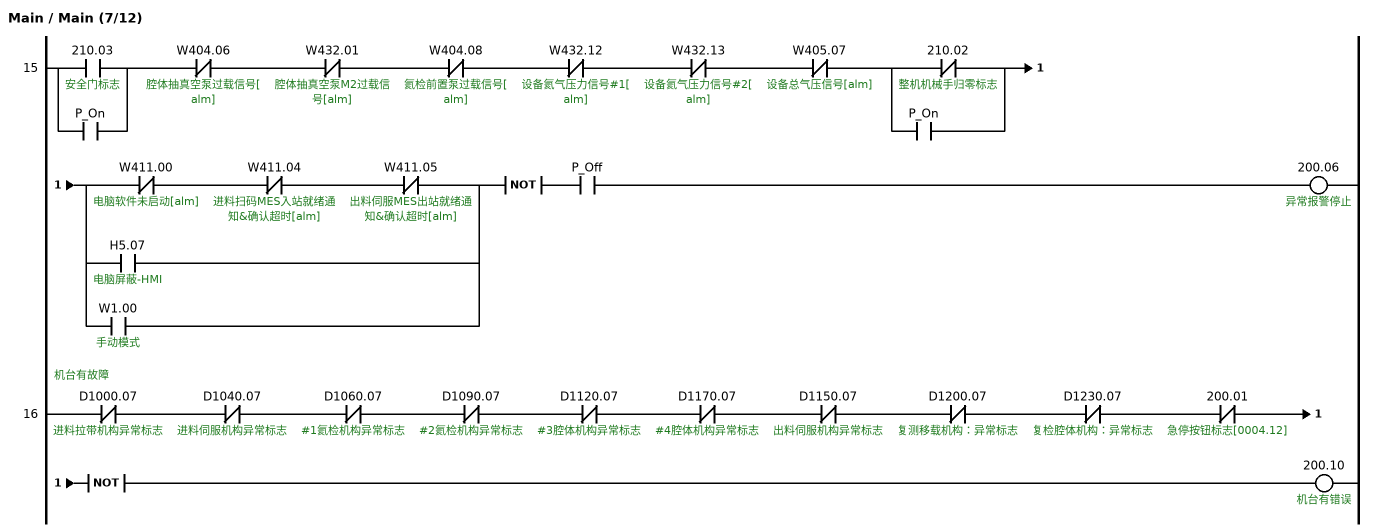
; rung 15
LD 210.03  ; 安全门标志
OR P_On
ANDNOT W404.06  ; 腔体抽真空泵过载信号[alm]
ANDNOT W432.01  ; 腔体抽真空泵M2过载信号[alm]
ANDNOT W404.08  ; 氦检前置泵过载信号[alm]
ANDNOT W432.12  ; 设备氦气压力信号#1[alm]
ANDNOT W432.13  ; 设备氦气压力信号#2[alm]
ANDNOT W405.07  ; 设备总气压信号[alm]
LDNOT 210.02  ; 整机机械手归零标志
OR P_On
ANDLD
LDNOT W411.00  ; 电脑软件未启动[alm]
ANDNOT W411.04  ; 进料扫码MES入站就绪通知&确认超时[alm]
ANDNOT W411.05  ; 出料伺服MES出站就绪通知&确认超时[alm]
OR H5.07  ; 电脑屏蔽-HMI
OR W1.00  ; 手动模式
ANDLD
NOT(520)
AND P_Off
OUT 200.06  ; 异常报警停止
; rung 16: 机台有故障
LDNOT D1000.07  ; 进料拉带机构异常标志
ANDNOT D1040.07  ; 进料伺服机构异常标志
ANDNOT D1060.07  ; #1氦检机构异常标志
ANDNOT D1090.07  ; #2氦检机构异常标志
ANDNOT D1120.07  ; #3腔体机构异常标志
ANDNOT D1170.07  ; #4腔体机构异常标志
ANDNOT D1150.07  ; 出料伺服机构异常标志
ANDNOT D1200.07  ; 复测移载机构：异常标志
ANDNOT D1230.07  ; 复检腔体机构：异常标志
ANDNOT 200.01  ; 急停按钮标志[0004.12]
NOT(520)
OUT 200.10  ; 机台有错误

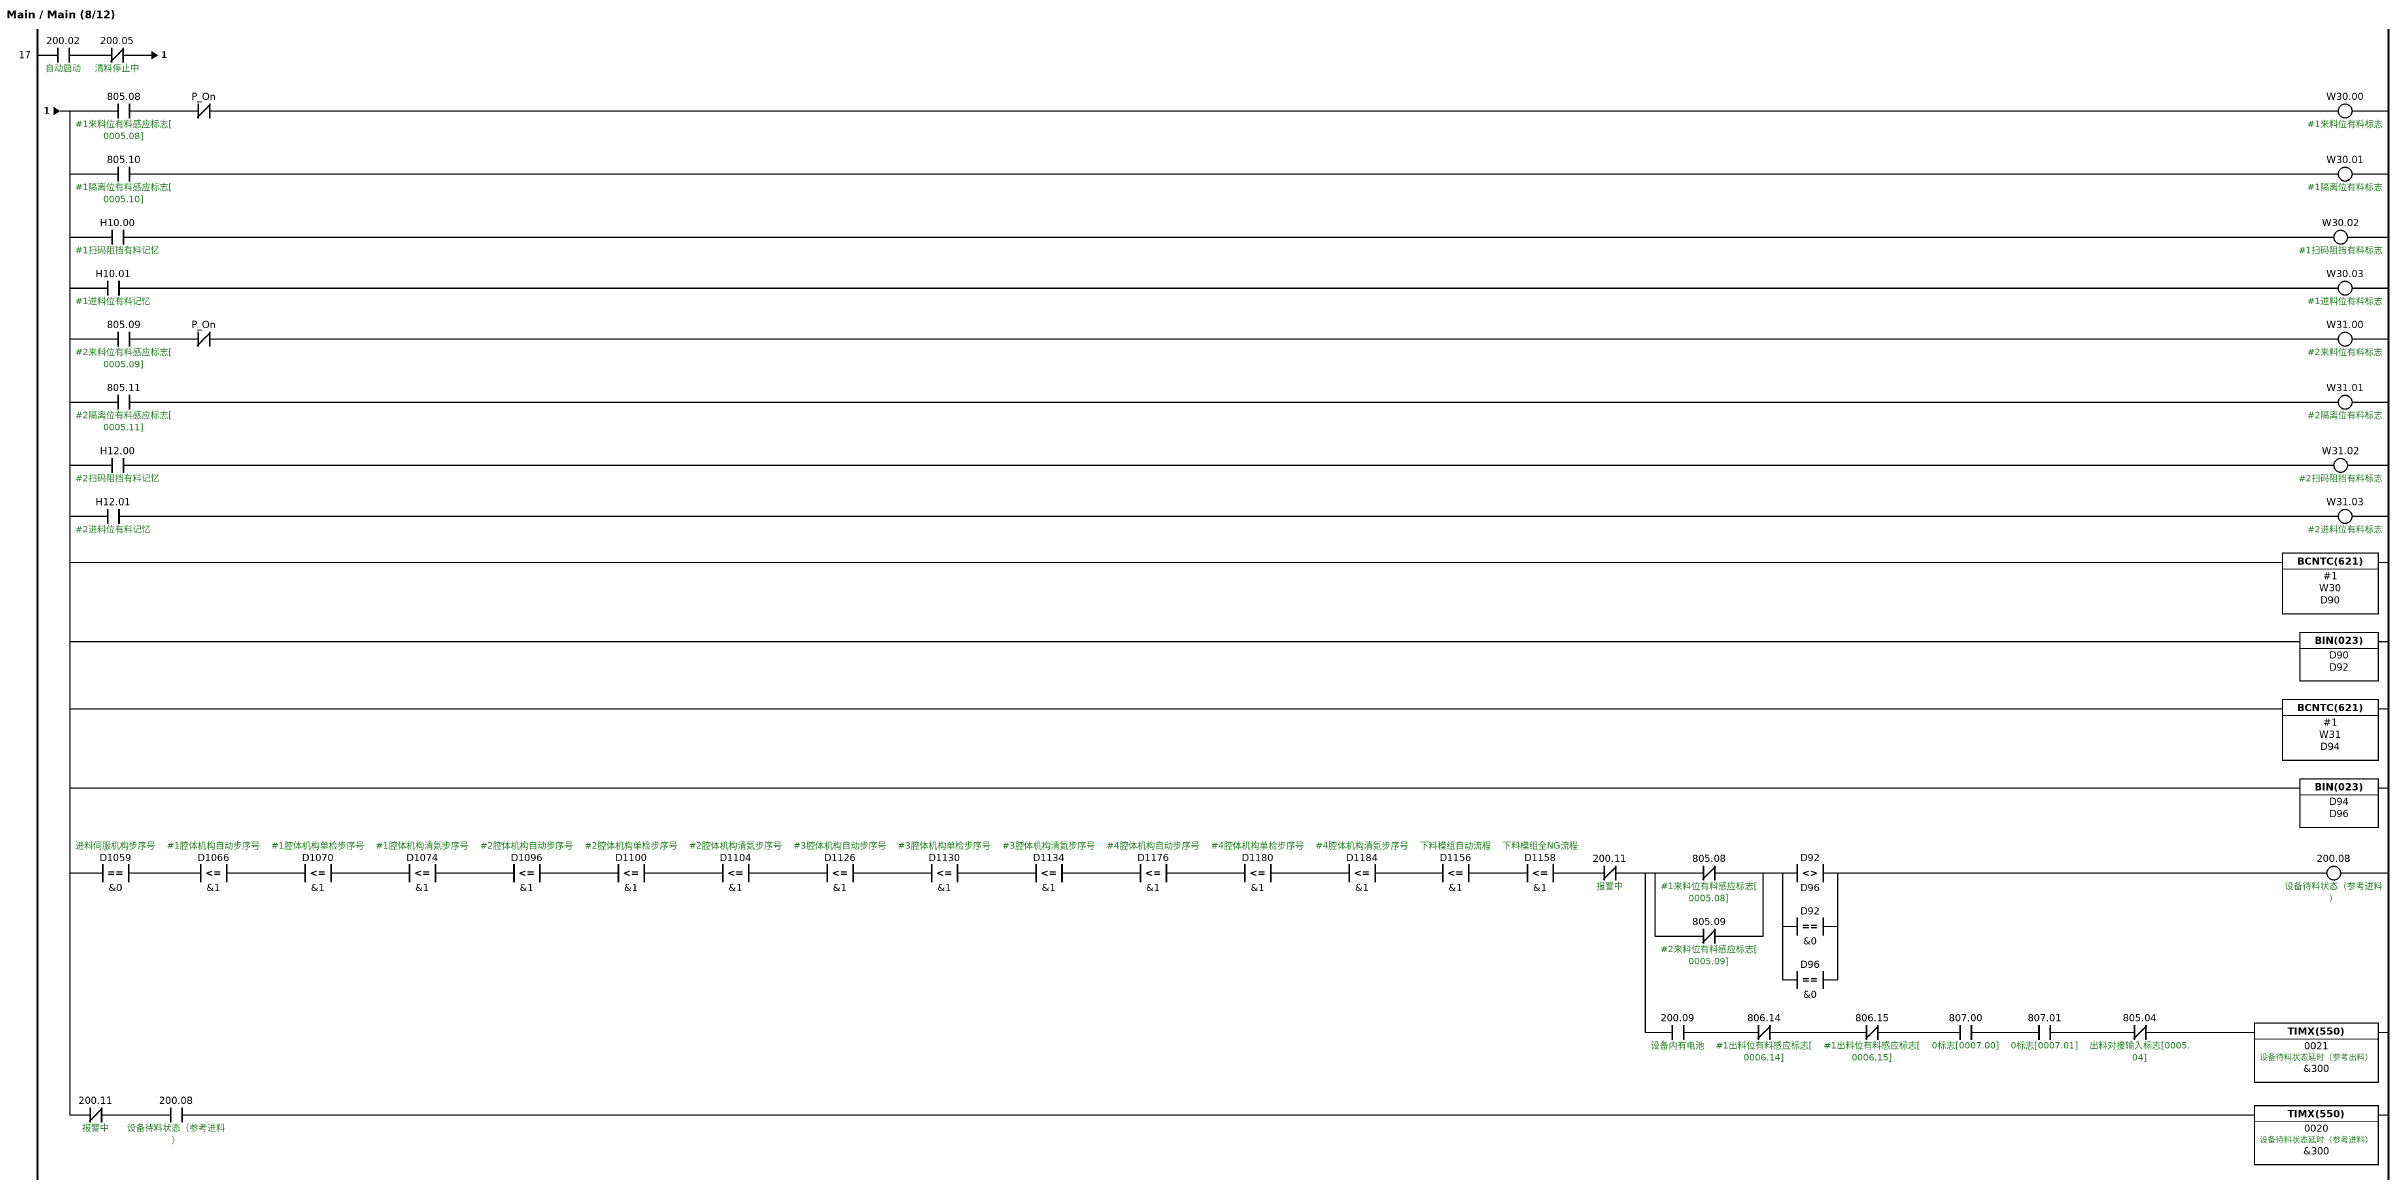
; rung 17
LD 200.02  ; 自动启动
ANDNOT 200.05  ; 清料停止中
OUT TR0
AND 805.08  ; #1来料位有料感应标志[0005.08]
ANDNOT P_On
OUT W30.00  ; #1来料位有料标志
LD TR0
AND 805.10  ; #1隔离位有料感应标志[0005.10]
OUT W30.01  ; #1隔离位有料标志
LD TR0
AND H10.00  ; #1扫码阻挡有料记忆
OUT W30.02  ; #1扫码阻挡有料标志
LD TR0
AND H10.01  ; #1进料位有料记忆
OUT W30.03  ; #1进料位有料标志
LD TR0
AND 805.09  ; #2来料位有料感应标志[0005.09]
ANDNOT P_On
OUT W31.00  ; #2来料位有料标志
LD TR0
AND 805.11  ; #2隔离位有料感应标志[0005.11]
OUT W31.01  ; #2隔离位有料标志
LD TR0
AND H12.00  ; #2扫码阻挡有料记忆
OUT W31.02  ; #2扫码阻挡有料标志
LD TR0
AND H12.01  ; #2进料位有料记忆
OUT W31.03  ; #2进料位有料标志
LD TR0
BCNTC(621) #1 W30 D90
BIN(023) D90 D92
BCNTC(621) #1 W31 D94
BIN(023) D94 D96
AND=(300) D1059 &0  ; 进料伺服机构步序号
AND<=L(316) D1066 &1  ; #1腔体机构自动步序号
AND<=L(316) D1070 &1  ; #1腔体机构单检步序号
AND<=L(316) D1074 &1  ; #1腔体机构清氦步序号
AND<=L(316) D1096 &1  ; #2腔体机构自动步序号
AND<=L(316) D1100 &1  ; #2腔体机构单检步序号
AND<=L(316) D1104 &1  ; #2腔体机构清氦步序号
AND<=L(316) D1126 &1  ; #3腔体机构自动步序号
AND<=L(316) D1130 &1  ; #3腔体机构单检步序号
AND<=L(316) D1134 &1  ; #3腔体机构清氦步序号
AND<=L(316) D1176 &1  ; #4腔体机构自动步序号
AND<=L(316) D1180 &1  ; #4腔体机构单检步序号
AND<=L(316) D1184 &1  ; #4腔体机构清氦步序号
AND<=L(316) D1156 &1  ; 下料模组自动流程
AND<=L(316) D1158 &1  ; 下料模组全NG流程
ANDNOT 200.11  ; 报警中
OUT TR1
LDNOT 805.08  ; #1来料位有料感应标志[0005.08]
ORNOT 805.09  ; #2来料位有料感应标志[0005.09]
ANDLD
LD<>(305) D92 D96
OR=(300) D92 &0
OR=(300) D96 &0
ANDLD
OUT 200.08  ; 设备待料状态（参考进料）
LD TR1
AND 200.09  ; 设备内有电池
ANDNOT 806.14  ; #1出料位有料感应标志[0006.14]
ANDNOT 806.15  ; #1出料位有料感应标志[0006.15]
AND 807.00  ; 0标志[0007.00]
AND 807.01  ; 0标志[0007.01]
ANDNOT 805.04  ; 出料对接输入标志[0005.04]
TIMX(550) 0021 &300  ; 设备待料状态延时（参考出料）
LD TR0
ANDNOT 200.11  ; 报警中
AND 200.08  ; 设备待料状态（参考进料）
TIMX(550) 0020 &300  ; 设备待料状态延时（参考进料）

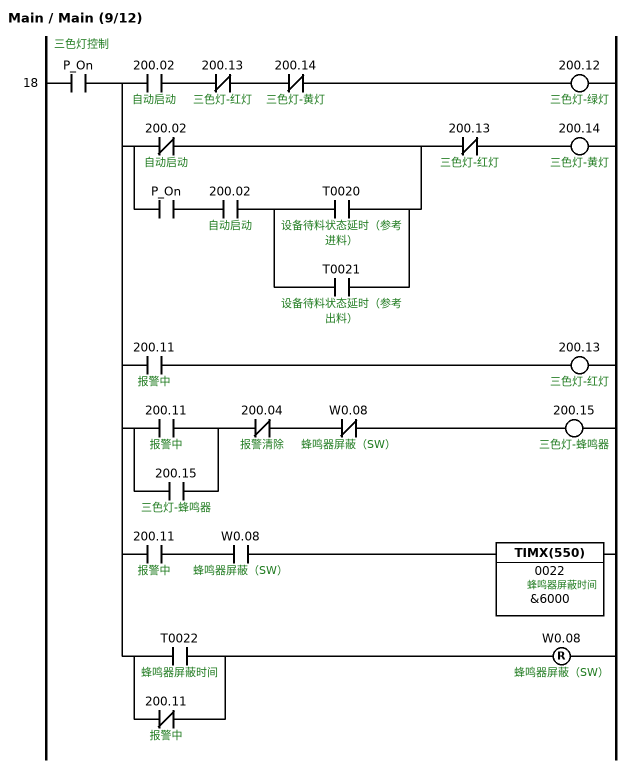
; rung 18: 三色灯控制
LD P_On
OUT TR0
AND 200.02  ; 自动启动
ANDNOT 200.13  ; 三色灯-红灯
ANDNOT 200.14  ; 三色灯-黄灯
OUT 200.12  ; 三色灯-绿灯
LD TR0
LDNOT 200.02  ; 自动启动
LD P_On
AND 200.02  ; 自动启动
LD T0020  ; 设备待料状态延时（参考进料）
OR T0021  ; 设备待料状态延时（参考出料）
ANDLD
ORLD
ANDLD
ANDNOT 200.13  ; 三色灯-红灯
OUT 200.14  ; 三色灯-黄灯
LD TR0
AND 200.11  ; 报警中
OUT 200.13  ; 三色灯-红灯
LD TR0
LD 200.11  ; 报警中
OR 200.15  ; 三色灯-蜂鸣器
ANDLD
ANDNOT 200.04  ; 报警清除
ANDNOT W0.08  ; 蜂鸣器屏蔽（SW）
OUT 200.15  ; 三色灯-蜂鸣器
LD TR0
AND 200.11  ; 报警中
AND W0.08  ; 蜂鸣器屏蔽（SW）
TIMX(550) 0022 &6000  ; 蜂鸣器屏蔽时间
LD TR0
LD T0022  ; 蜂鸣器屏蔽时间
ORNOT 200.11  ; 报警中
ANDLD
RSET W0.08  ; 蜂鸣器屏蔽（SW）

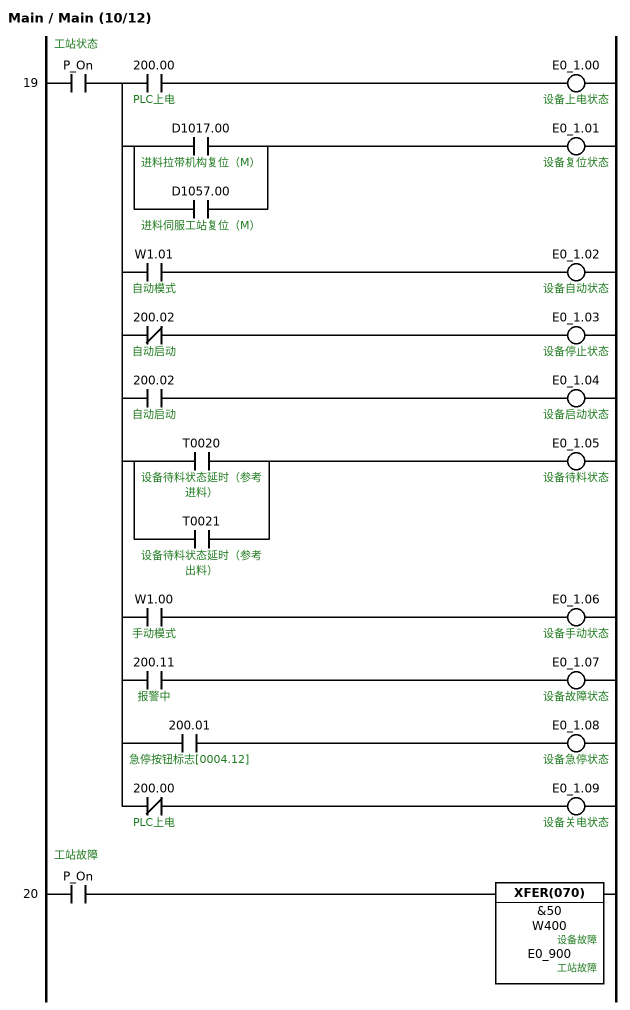
; rung 19: 工站状态
LD P_On
OUT TR0
AND 200.00  ; PLC上电
OUT E0_1.00  ; 设备上电状态
LD TR0
LD D1017.00  ; 进料拉带机构复位（M）
OR D1057.00  ; 进料伺服工站复位（M）
ANDLD
OUT E0_1.01  ; 设备复位状态
LD TR0
AND W1.01  ; 自动模式
OUT E0_1.02  ; 设备自动状态
LD TR0
ANDNOT 200.02  ; 自动启动
OUT E0_1.03  ; 设备停止状态
LD TR0
AND 200.02  ; 自动启动
OUT E0_1.04  ; 设备启动状态
LD TR0
LD T0020  ; 设备待料状态延时（参考进料）
OR T0021  ; 设备待料状态延时（参考出料）
ANDLD
OUT E0_1.05  ; 设备待料状态
LD TR0
AND W1.00  ; 手动模式
OUT E0_1.06  ; 设备手动状态
LD TR0
AND 200.11  ; 报警中
OUT E0_1.07  ; 设备故障状态
LD TR0
AND 200.01  ; 急停按钮标志[0004.12]
OUT E0_1.08  ; 设备急停状态
LD TR0
ANDNOT 200.00  ; PLC上电
OUT E0_1.09  ; 设备关电状态
; rung 20: 工站故障
LD P_On
XFER(070) &50 W400 E0_900  ; 设备故障, 工站故障

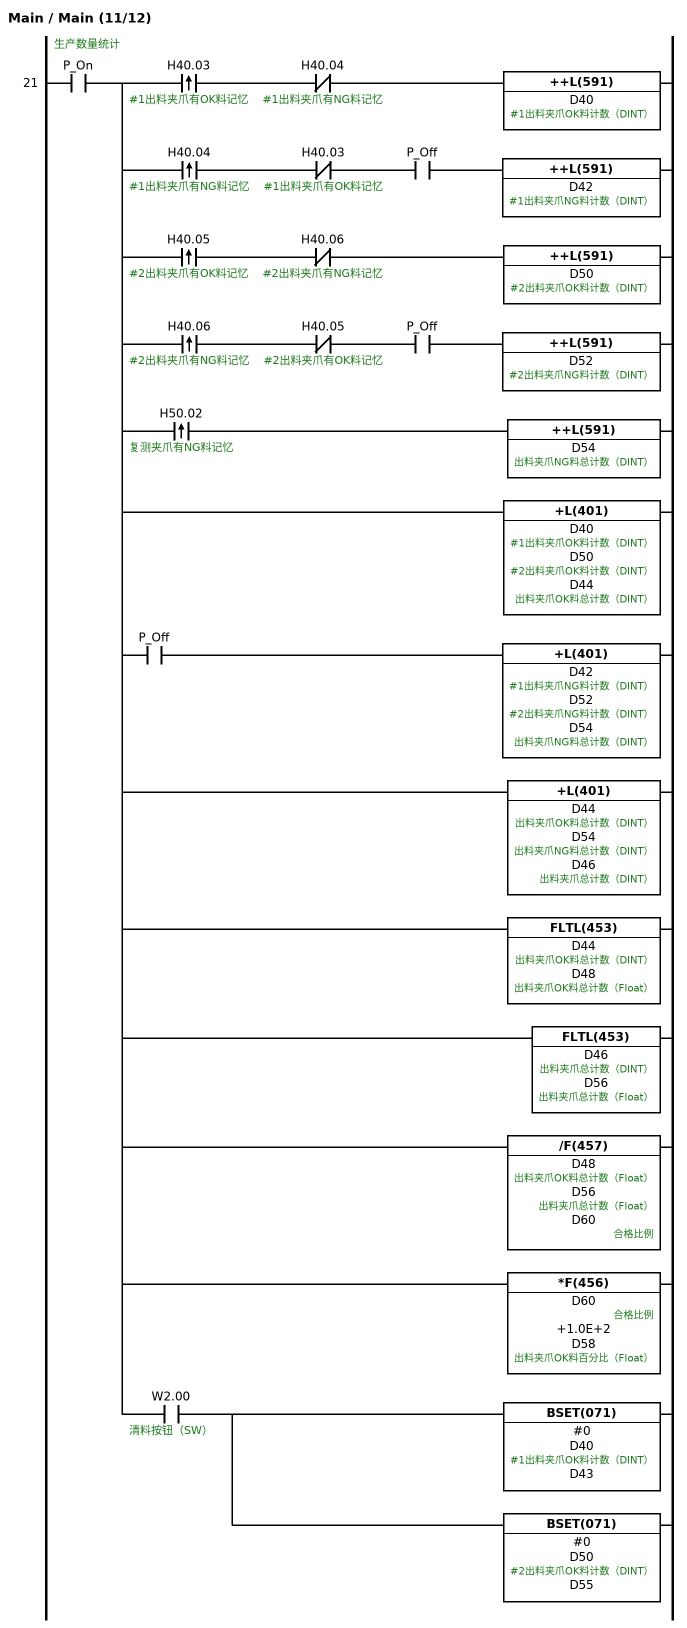
; rung 21: 生产数量统计
LD P_On
OUT TR0
@AND H40.03  ; #1出料夹爪有OK料记忆
ANDNOT H40.04  ; #1出料夹爪有NG料记忆
++L(591) D40  ; #1出料夹爪OK料计数（DINT）
LD TR0
@AND H40.04  ; #1出料夹爪有NG料记忆
ANDNOT H40.03  ; #1出料夹爪有OK料记忆
AND P_Off
++L(591) D42  ; #1出料夹爪NG料计数（DINT）
LD TR0
@AND H40.05  ; #2出料夹爪有OK料记忆
ANDNOT H40.06  ; #2出料夹爪有NG料记忆
++L(591) D50  ; #2出料夹爪OK料计数（DINT）
LD TR0
@AND H40.06  ; #2出料夹爪有NG料记忆
ANDNOT H40.05  ; #2出料夹爪有OK料记忆
AND P_Off
++L(591) D52  ; #2出料夹爪NG料计数（DINT）
LD TR0
@AND H50.02  ; 复测夹爪有NG料记忆
++L(591) D54  ; 出料夹爪NG料总计数（DINT）
LD TR0
+L(401) D40 D50 D44  ; #1出料夹爪OK料计数（DINT）, #2出料夹爪OK料计数（DINT）, 出料夹爪OK料总计数（DINT）
AND P_Off
+L(401) D42 D52 D54  ; #1出料夹爪NG料计数（DINT）, #2出料夹爪NG料计数（DINT）, 出料夹爪NG料总计数（DINT）
LD TR0
+L(401) D44 D54 D46  ; 出料夹爪OK料总计数（DINT）, 出料夹爪NG料总计数（DINT）, 出料夹爪总计数（DINT）
FLTL(453) D44 D48  ; 出料夹爪OK料总计数（DINT）, 出料夹爪OK料总计数（Float）
FLTL(453) D46 D56  ; 出料夹爪总计数（DINT）, 出料夹爪总计数（Float）
/F(457) D48 D56 D60  ; 出料夹爪OK料总计数（Float）, 出料夹爪总计数（Float）, 合格比例
*F(456) D60 +1.0E+2 D58  ; 合格比例, 出料夹爪OK料百分比（Float）
AND W2.00  ; 清料按钮（SW）
BSET(071) #0 D40 D43  ; #1出料夹爪OK料计数（DINT）
BSET(071) #0 D50 D55  ; #2出料夹爪OK料计数（DINT）

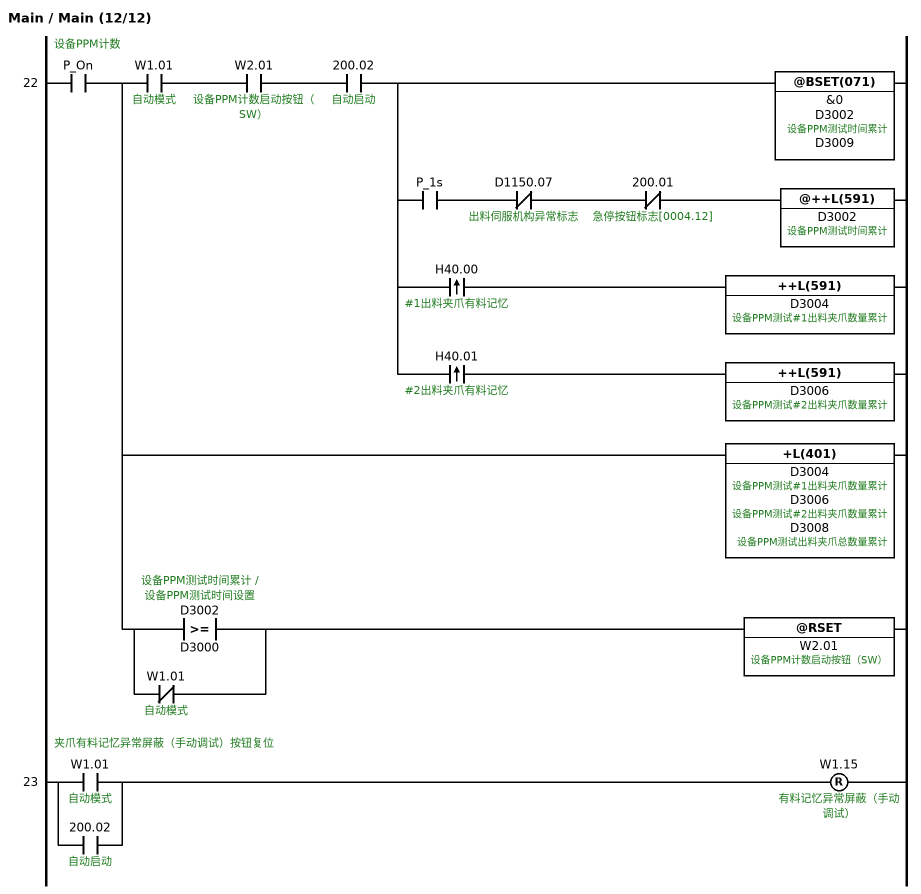
; rung 22: 设备PPM计数
LD P_On
OUT TR0
AND W1.01  ; 自动模式
AND W2.01  ; 设备PPM计数启动按钮（SW）  // HMI《切换开关》按钮
AND 200.02  ; 自动启动
OUT TR1
@BSET(071) &0 D3002 D3009  ; 设备PPM测试时间累计
AND P_1s
ANDNOT D1150.07  ; 出料伺服机构异常标志
ANDNOT 200.01  ; 急停按钮标志[0004.12]
@++L(591) D3002  ; 设备PPM测试时间累计
LD TR1
@AND H40.00  ; #1出料夹爪有料记忆
++L(591) D3004  ; 设备PPM测试#1出料夹爪数量累计
LD TR1
@AND H40.01  ; #2出料夹爪有料记忆
++L(591) D3006  ; 设备PPM测试#2出料夹爪数量累计
LD TR0
+L(401) D3004 D3006 D3008  ; 设备PPM测试#1出料夹爪数量累计, 设备PPM测试#2出料夹爪数量累计, 设备PPM测试出料夹爪总数量累计
LD>=L(326) D3002 D3000  ; 设备PPM测试时间累计, 设备PPM测试时间设置
ORNOT W1.01  ; 自动模式
ANDLD
@RSET W2.01  ; 设备PPM计数启动按钮（SW）
; rung 23: 夹爪有料记忆异常屏蔽（手动调试）按钮复位
LD W1.01  ; 自动模式
OR 200.02  ; 自动启动
RSET W1.15  ; 有料记忆异常屏蔽（手动调试）
; rung 24: 对接信号

### Section 氦检仪通讯

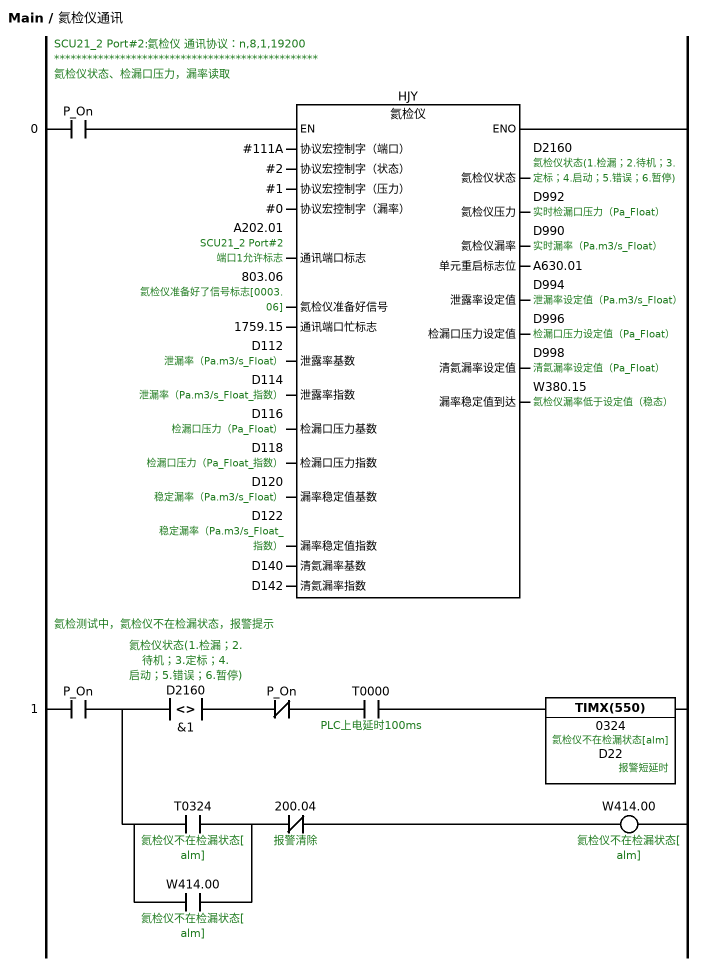
; rung 0: SCU21_2 Port#2:氦检仪 通讯协议：n,8,1,19200 / ************************************************ / 氦检仪状态、检漏口压力，漏率读取
LD P_On
CALL HJY : 氦检仪 (协议宏控制字（端口） := #111A, 协议宏控制字（状态） := #2, 协议宏控制字（压力） := #1, 协议宏控制字（漏率） := #0, 通讯端口标志 := A202.01, 氦检仪准备好信号 := 803.06, 通讯端口忙标志 := 1759.15, 泄露率基数 := D112, 泄露率指数 := D114, 检漏口压力基数 := D116, 检漏口压力指数 := D118, 漏率稳定值基数 := D120, 漏率稳定值指数 := D122, 清氦漏率基数 := D140, 清氦漏率指数 := D142, 氦检仪状态 => D2160, 氦检仪压力 => D992, 氦检仪漏率 => D990, 单元重启标志位 => A630.01, 泄露率设定值 => D994, 检漏口压力设定值 => D996, 清氦漏率设定值 => D998, 漏率稳定值到达 => W380.15)  ; SCU21_2 Port#2 端口1允许标志, 氦检仪准备好了信号标志[0003.06], 泄漏率（Pa.m3/s_Float）, 泄漏率（Pa.m3/s_Float_指数）, 检漏口压力（Pa_Float）, 检漏口压力（Pa_Float_指数）, 稳定漏率（Pa.m3/s_Float）, 稳定漏率（Pa.m3/s_Float_指数）, 氦检仪状态(1.检漏；2.待机；3.定标；4.启动；5.错误；6.暂停), 实时检漏口压力（Pa_Float）, 实时漏率（Pa.m3/s_Float）, 泄漏率设定值（Pa.m3/s_Float）, 检漏口压力设定值（Pa_Float）, 清氦漏率设定值（Pa_Float）, 氦检仪漏率低于设定值（稳态）
; rung 1: 氦检测试中，氦检仪不在检漏状态，报警提示
LD P_On
OUT TR0
AND<>(305) D2160 &1  ; 氦检仪状态(1.检漏；2.待机；3.定标；4.启动；5.错误；6.暂停)
ANDNOT P_On  // 各腔体氦检步DXXXX.00=1
AND T0000  ; PLC上电延时100ms
TIMX(550) 0324 D22  ; 报警短延时, 氦检仪不在检漏状态[alm]
LD TR0
LD T0324  ; 氦检仪不在检漏状态[alm]
OR W414.00  ; 氦检仪不在检漏状态[alm]
ANDLD
ANDNOT 200.04  ; 报警清除
OUT W414.00  ; 氦检仪不在检漏状态[alm]

### Section 入料扫码通讯

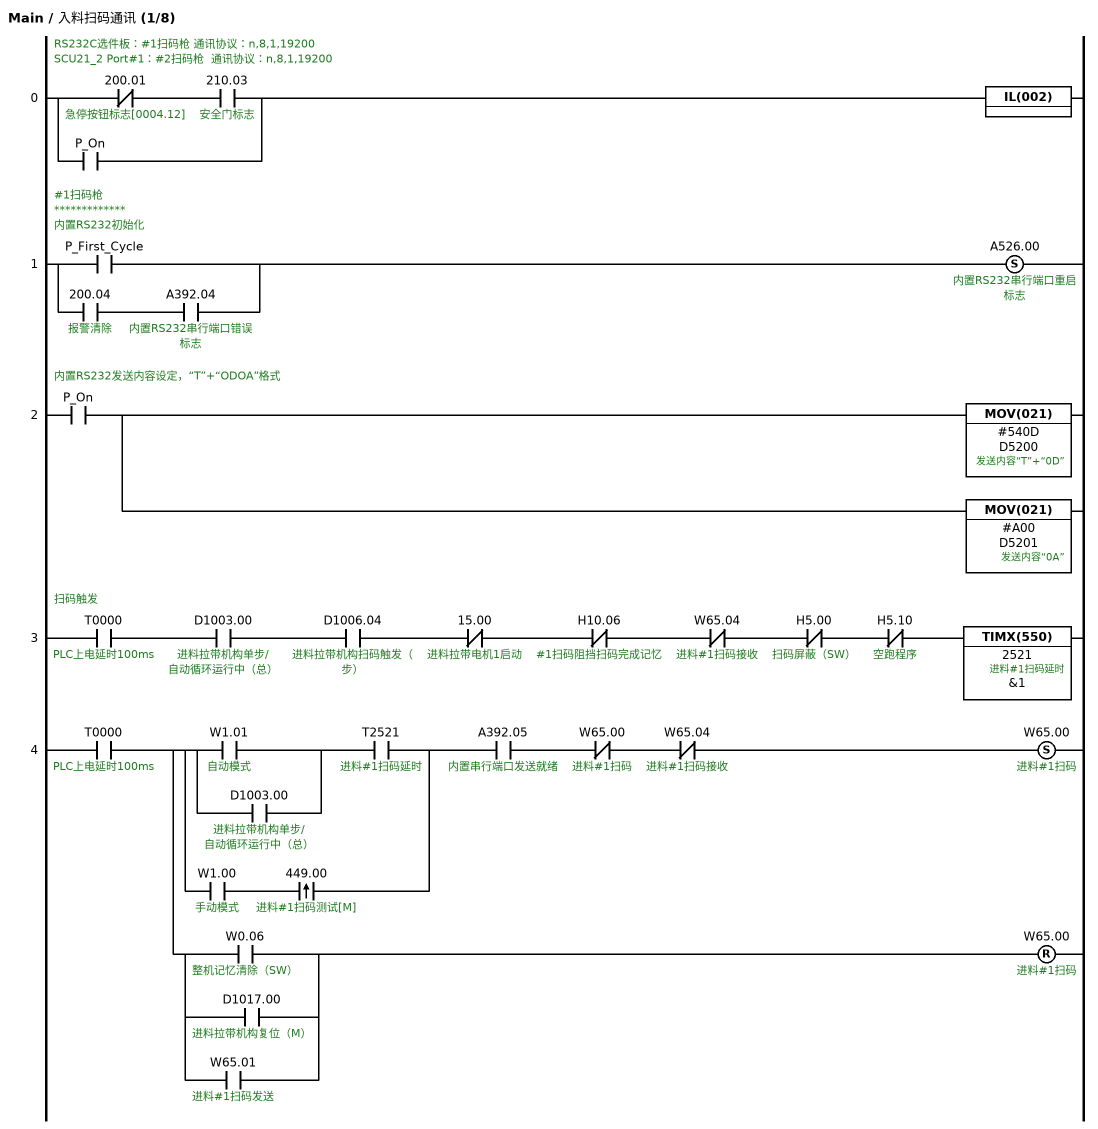
; rung 0: RS232C选件板：#1扫码枪 通讯协议：n,8,1,19200 / SCU21_2 Port#1：#2扫码枪  通讯协议：n,8,1,19200
LDNOT 200.01  ; 急停按钮标志[0004.12]
AND 210.03  ; 安全门标志
OR P_On
IL(002)
; rung 1: #1扫码枪 / ************* / 内置RS232初始化
LD P_First_Cycle
LD 200.04  ; 报警清除
AND A392.04  ; 内置RS232串行端口错误标志
ORLD
SET A526.00  ; 内置RS232串行端口重启标志
; rung 2: 内置RS232发送内容设定，“T”+“ODOA”格式
LD P_On
MOV(021) #540D D5200  ; 发送内容“T”+“0D”
MOV(021) #A00 D5201  ; 发送内容“0A”
; rung 3: 扫码触发
LD T0000  ; PLC上电延时100ms
AND D1003.00  ; 进料拉带机构单步/自动循环运行中（总）
AND D1006.04  ; 进料拉带机构扫码触发（步）
ANDNOT 15.00  ; 进料拉带电机1启动
ANDNOT H10.06  ; #1扫码阻挡扫码完成记忆
ANDNOT W65.04  ; 进料#1扫码接收
ANDNOT H5.00  ; 扫码屏蔽（SW）
ANDNOT H5.10  ; 空跑程序
TIMX(550) 2521 &1  ; 进料#1扫码延时
; rung 4
LD T0000  ; PLC上电延时100ms
OUT TR0
LD W1.01  ; 自动模式
OR D1003.00  ; 进料拉带机构单步/自动循环运行中（总）
AND T2521  ; 进料#1扫码延时
LD W1.00  ; 手动模式
@AND 449.00  ; 进料#1扫码测试[M]
ORLD
ANDLD
AND A392.05  ; 内置串行端口发送就绪
ANDNOT W65.00  ; 进料#1扫码
ANDNOT W65.04  ; 进料#1扫码接收
SET W65.00  ; 进料#1扫码
LD TR0
LD W0.06  ; 整机记忆清除（SW）
OR D1017.00  ; 进料拉带机构复位（M）
OR W65.01  ; 进料#1扫码发送
ANDLD
RSET W65.00  ; 进料#1扫码

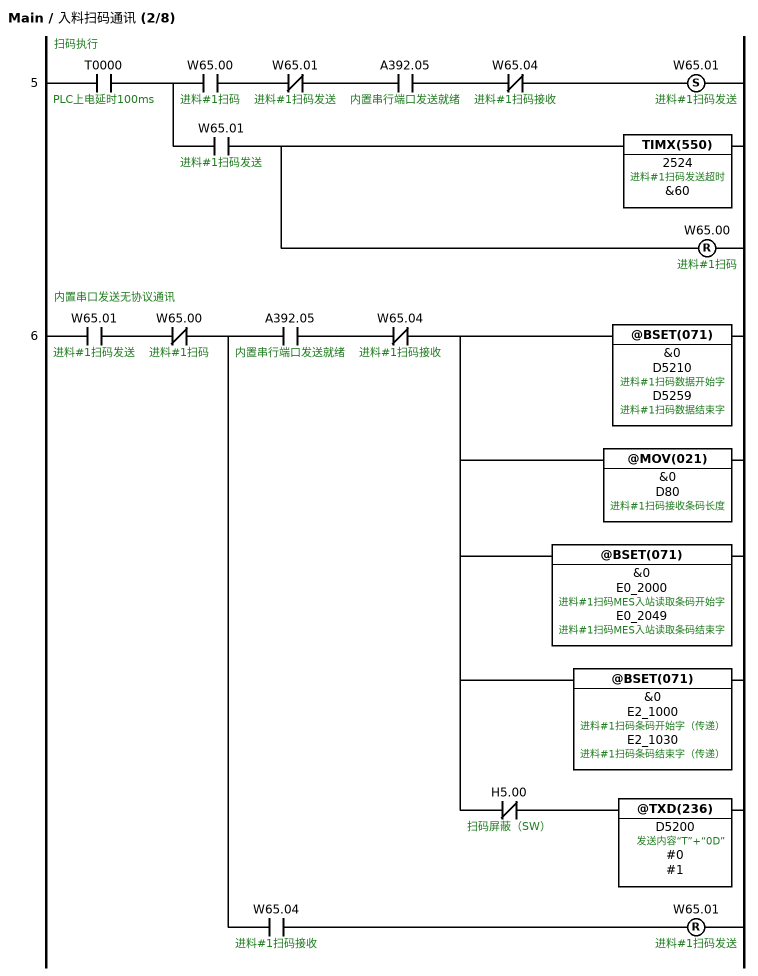
; rung 5: 扫码执行
LD T0000  ; PLC上电延时100ms
OUT TR0
AND W65.00  ; 进料#1扫码
ANDNOT W65.01  ; 进料#1扫码发送
AND A392.05  ; 内置串行端口发送就绪
ANDNOT W65.04  ; 进料#1扫码接收
SET W65.01  ; 进料#1扫码发送
LD TR0
AND W65.01  ; 进料#1扫码发送
TIMX(550) 2524 &60  ; 进料#1扫码发送超时
RSET W65.00  ; 进料#1扫码
; rung 6: 内置串口发送无协议通讯
LD W65.01  ; 进料#1扫码发送
ANDNOT W65.00  ; 进料#1扫码
OUT TR0
AND A392.05  ; 内置串行端口发送就绪
ANDNOT W65.04  ; 进料#1扫码接收
@BSET(071) &0 D5210 D5259  ; 进料#1扫码数据开始字, 进料#1扫码数据结束字
@MOV(021) &0 D80  ; 进料#1扫码接收条码长度
@BSET(071) &0 E0_2000 E0_2049  ; 进料#1扫码MES入站读取条码开始字, 进料#1扫码MES入站读取条码结束字
@BSET(071) &0 E2_1000 E2_1030  ; 进料#1扫码条码开始字（传递）, 进料#1扫码条码结束字（传递）
ANDNOT H5.00  ; 扫码屏蔽（SW）
@TXD(236) D5200 #0 #1  ; 发送内容“T”+“0D”
LD TR0
AND W65.04  ; 进料#1扫码接收
RSET W65.01  ; 进料#1扫码发送

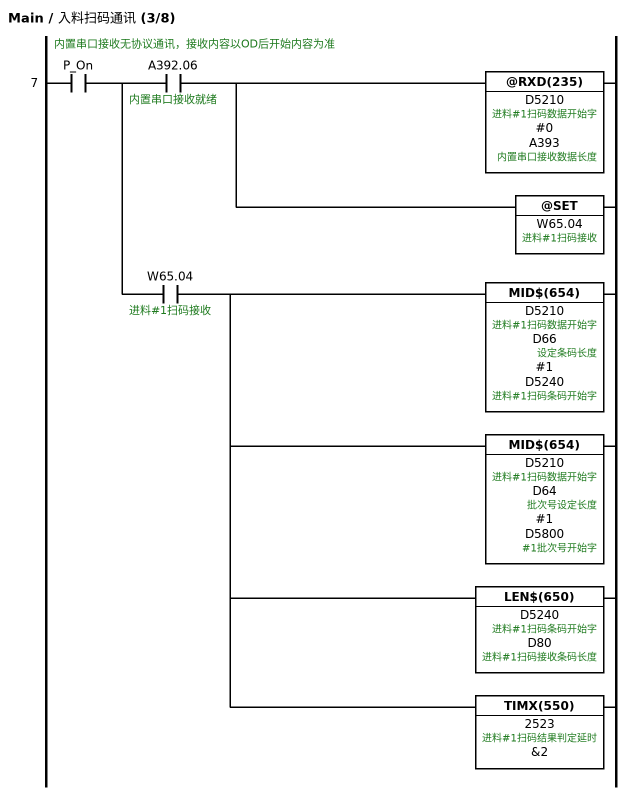
; rung 7: 内置串口接收无协议通讯，接收内容以OD后开始内容为准
LD P_On
OUT TR0
AND A392.06  ; 内置串口接收就绪
@RXD(235) D5210 #0 A393  ; 进料#1扫码数据开始字, 内置串口接收数据长度
@SET W65.04  ; 进料#1扫码接收
LD TR0
AND W65.04  ; 进料#1扫码接收
MID$(654) D5210 D66 #1 D5240  ; 进料#1扫码数据开始字, 设定条码长度, 进料#1扫码条码开始字
MID$(654) D5210 D64 #1 D5800  ; 进料#1扫码数据开始字, 批次号设定长度, #1批次号开始字
LEN$(650) D5240 D80  ; 进料#1扫码条码开始字, 进料#1扫码接收条码长度
TIMX(550) 2523 &2  ; 进料#1扫码结果判定延时

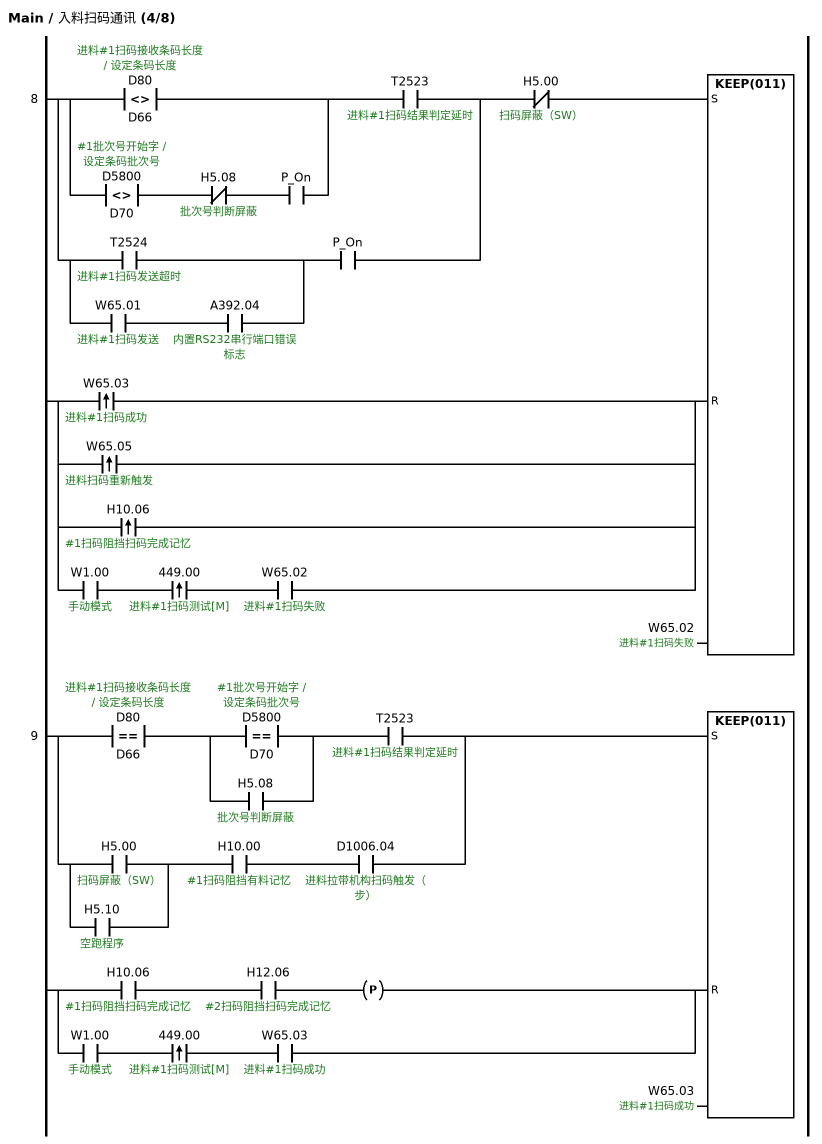
; rung 8
LD<>(305) D80 D66  ; 进料#1扫码接收条码长度, 设定条码长度
LD<>$(671) D5800 D70  ; #1批次号开始字, 设定条码批次号
ANDNOT H5.08  ; 批次号判断屏蔽
AND P_On
ORLD
AND T2523  ; 进料#1扫码结果判定延时
LD T2524  ; 进料#1扫码发送超时
LD W65.01  ; 进料#1扫码发送
AND A392.04  ; 内置RS232串行端口错误标志
ORLD
AND P_On
ORLD
ANDNOT H5.00  ; 扫码屏蔽（SW）
@LD W65.03  ; 进料#1扫码成功
@OR W65.05  ; 进料扫码重新触发
@OR H10.06  ; #1扫码阻挡扫码完成记忆
LD W1.00  ; 手动模式
@AND 449.00  ; 进料#1扫码测试[M]
AND W65.02  ; 进料#1扫码失败
ORLD
KEEP(011) W65.02  ; 进料#1扫码失败
; rung 9
LD=(300) D80 D66  ; 进料#1扫码接收条码长度, 设定条码长度
LD=$(670) D5800 D70  ; #1批次号开始字, 设定条码批次号
OR H5.08  ; 批次号判断屏蔽
ANDLD
AND T2523  ; 进料#1扫码结果判定延时
LD H5.00  ; 扫码屏蔽（SW）
OR H5.10  ; 空跑程序
AND H10.00  ; #1扫码阻挡有料记忆
AND D1006.04  ; 进料拉带机构扫码触发（步）
ORLD
LD H10.06  ; #1扫码阻挡扫码完成记忆
AND H12.06  ; #2扫码阻挡扫码完成记忆
UP(521)
LD W1.00  ; 手动模式
@AND 449.00  ; 进料#1扫码测试[M]
AND W65.03  ; 进料#1扫码成功
ORLD
KEEP(011) W65.03  ; 进料#1扫码成功

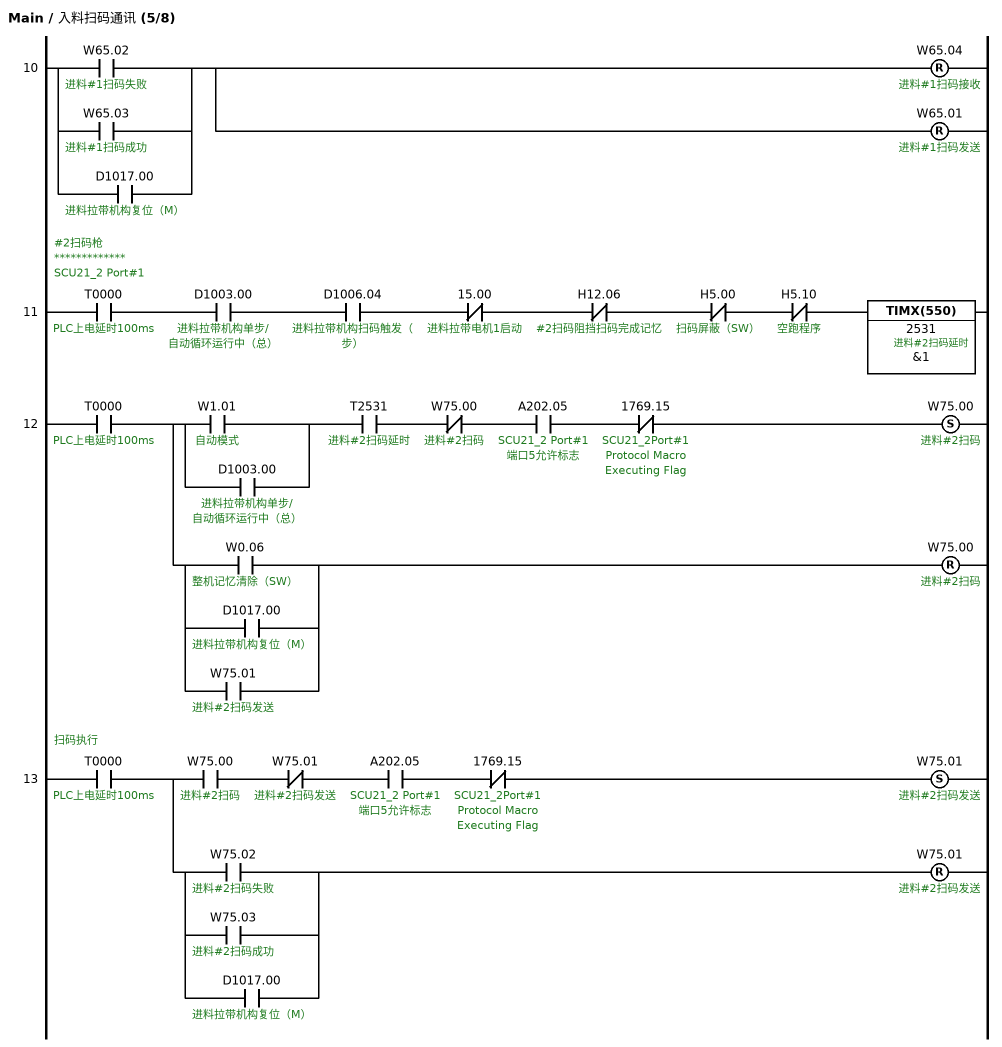
; rung 10
LD W65.02  ; 进料#1扫码失败
OR W65.03  ; 进料#1扫码成功
OR D1017.00  ; 进料拉带机构复位（M）
RSET W65.04  ; 进料#1扫码接收
RSET W65.01  ; 进料#1扫码发送
; rung 11: #2扫码枪 / ************* / SCU21_2 Port#1
LD T0000  ; PLC上电延时100ms
AND D1003.00  ; 进料拉带机构单步/自动循环运行中（总）
AND D1006.04  ; 进料拉带机构扫码触发（步）
ANDNOT 15.00  ; 进料拉带电机1启动
ANDNOT H12.06  ; #2扫码阻挡扫码完成记忆
ANDNOT H5.00  ; 扫码屏蔽（SW）
ANDNOT H5.10  ; 空跑程序
TIMX(550) 2531 &1  ; 进料#2扫码延时
; rung 12
LD T0000  ; PLC上电延时100ms
OUT TR0
LD W1.01  ; 自动模式
OR D1003.00  ; 进料拉带机构单步/自动循环运行中（总）
ANDLD
AND T2531  ; 进料#2扫码延时
ANDNOT W75.00  ; 进料#2扫码
AND A202.05  ; SCU21_2 Port#1 端口5允许标志
ANDNOT 1769.15  ; SCU21_2Port#1 Protocol Macro Executing Flag
SET W75.00  ; 进料#2扫码
LD TR0
LD W0.06  ; 整机记忆清除（SW）
OR D1017.00  ; 进料拉带机构复位（M）
OR W75.01  ; 进料#2扫码发送
ANDLD
RSET W75.00  ; 进料#2扫码
; rung 13: 扫码执行
LD T0000  ; PLC上电延时100ms
OUT TR0
AND W75.00  ; 进料#2扫码
ANDNOT W75.01  ; 进料#2扫码发送
AND A202.05  ; SCU21_2 Port#1 端口5允许标志
ANDNOT 1769.15  ; SCU21_2Port#1 Protocol Macro Executing Flag
SET W75.01  ; 进料#2扫码发送
LD TR0
LD W75.02  ; 进料#2扫码失败
OR W75.03  ; 进料#2扫码成功
OR D1017.00  ; 进料拉带机构复位（M）
ANDLD
RSET W75.01  ; 进料#2扫码发送

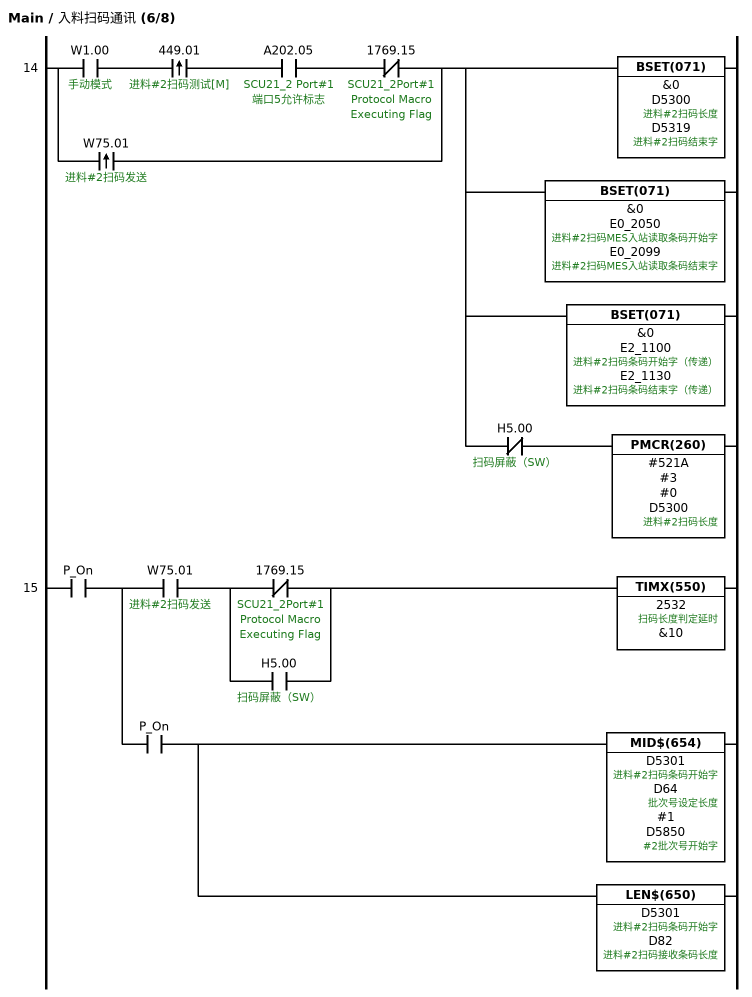
; rung 14
LD W1.00  ; 手动模式
@AND 449.01  ; 进料#2扫码测试[M]
AND A202.05  ; SCU21_2 Port#1 端口5允许标志
ANDNOT 1769.15  ; SCU21_2Port#1 Protocol Macro Executing Flag
@OR W75.01  ; 进料#2扫码发送
BSET(071) &0 D5300 D5319  ; 进料#2扫码长度, 进料#2扫码结束字
BSET(071) &0 E0_2050 E0_2099  ; 进料#2扫码MES入站读取条码开始字, 进料#2扫码MES入站读取条码结束字
BSET(071) &0 E2_1100 E2_1130  ; 进料#2扫码条码开始字（传递）, 进料#2扫码条码结束字（传递）
ANDNOT H5.00  ; 扫码屏蔽（SW）
PMCR(260) #521A #3 #0 D5300  ; 进料#2扫码长度
; rung 15
LD P_On
OUT TR0
AND W75.01  ; 进料#2扫码发送
LDNOT 1769.15  ; SCU21_2Port#1 Protocol Macro Executing Flag
OR H5.00  ; 扫码屏蔽（SW）
ANDLD
TIMX(550) 2532 &10  ; 扫码长度判定延时
LD TR0
AND P_On
MID$(654) D5301 D64 #1 D5850  ; 进料#2扫码条码开始字, 批次号设定长度, #2批次号开始字
LEN$(650) D5301 D82  ; 进料#2扫码条码开始字, 进料#2扫码接收条码长度

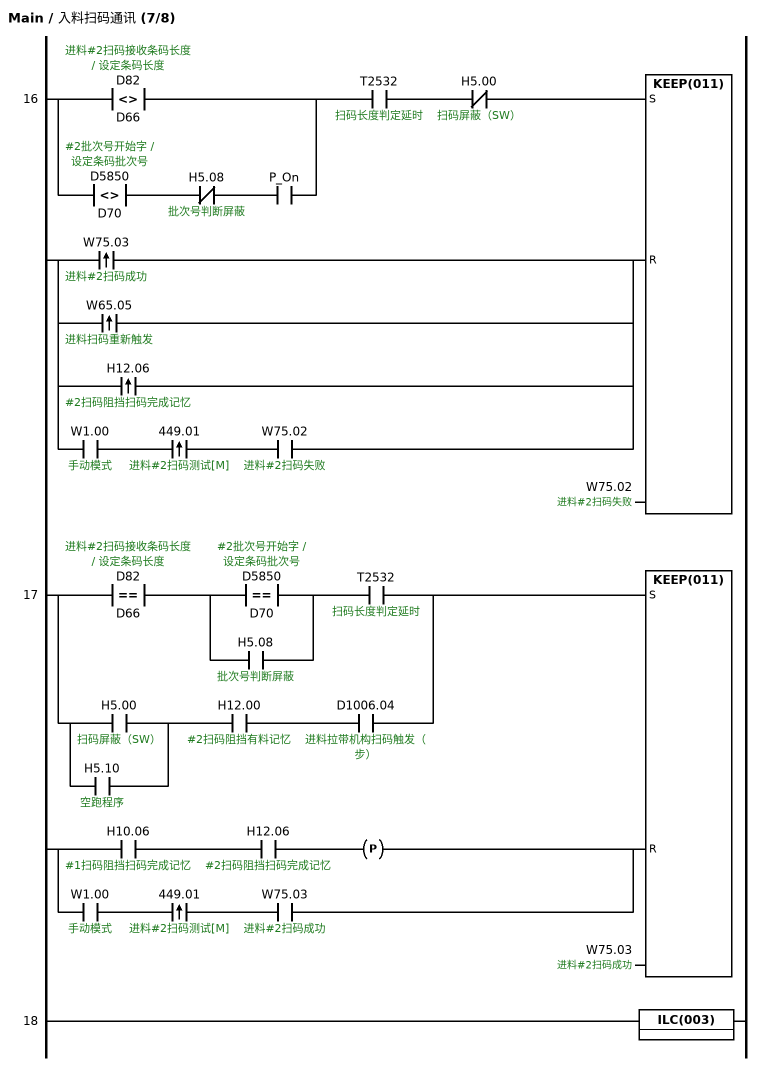
; rung 16
LD<>(305) D82 D66  ; 进料#2扫码接收条码长度, 设定条码长度
LD<>$(671) D5850 D70  ; #2批次号开始字, 设定条码批次号
ANDNOT H5.08  ; 批次号判断屏蔽
AND P_On
ORLD
AND T2532  ; 扫码长度判定延时
ANDNOT H5.00  ; 扫码屏蔽（SW）
@LD W75.03  ; 进料#2扫码成功
@OR W65.05  ; 进料扫码重新触发
@OR H12.06  ; #2扫码阻挡扫码完成记忆
LD W1.00  ; 手动模式
@AND 449.01  ; 进料#2扫码测试[M]
AND W75.02  ; 进料#2扫码失败
ORLD
KEEP(011) W75.02  ; 进料#2扫码失败
; rung 17
LD=(300) D82 D66  ; 进料#2扫码接收条码长度, 设定条码长度
LD=$(670) D5850 D70  ; #2批次号开始字, 设定条码批次号
OR H5.08  ; 批次号判断屏蔽
ANDLD
AND T2532  ; 扫码长度判定延时
LD H5.00  ; 扫码屏蔽（SW）
OR H5.10  ; 空跑程序
AND H12.00  ; #2扫码阻挡有料记忆
AND D1006.04  ; 进料拉带机构扫码触发（步）
ORLD
LD H10.06  ; #1扫码阻挡扫码完成记忆
AND H12.06  ; #2扫码阻挡扫码完成记忆
UP(521)
LD W1.00  ; 手动模式
@AND 449.01  ; 进料#2扫码测试[M]
AND W75.03  ; 进料#2扫码成功
ORLD
KEEP(011) W75.03  ; 进料#2扫码成功
; rung 18
ILC(003)

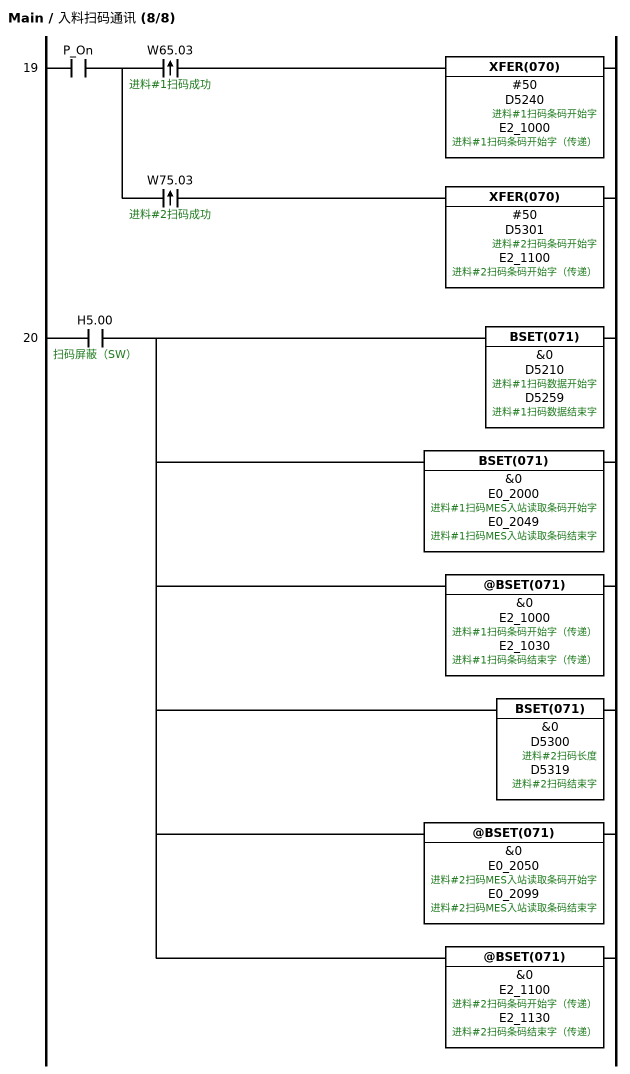
; rung 19
LD P_On
OUT TR0
@AND W65.03  ; 进料#1扫码成功
XFER(070) #50 D5240 E2_1000  ; 进料#1扫码条码开始字, 进料#1扫码条码开始字（传递）
LD TR0
@AND W75.03  ; 进料#2扫码成功
XFER(070) #50 D5301 E2_1100  ; 进料#2扫码条码开始字, 进料#2扫码条码开始字（传递）
; rung 20
LD H5.00  ; 扫码屏蔽（SW）
BSET(071) &0 D5210 D5259  ; 进料#1扫码数据开始字, 进料#1扫码数据结束字
BSET(071) &0 E0_2000 E0_2049  ; 进料#1扫码MES入站读取条码开始字, 进料#1扫码MES入站读取条码结束字
@BSET(071) &0 E2_1000 E2_1030  ; 进料#1扫码条码开始字（传递）, 进料#1扫码条码结束字（传递）
BSET(071) &0 D5300 D5319  ; 进料#2扫码长度, 进料#2扫码结束字
@BSET(071) &0 E0_2050 E0_2099  ; 进料#2扫码MES入站读取条码开始字, 进料#2扫码MES入站读取条码结束字
@BSET(071) &0 E2_1100 E2_1130  ; 进料#2扫码条码开始字（传递）, 进料#2扫码条码结束字（传递）

### Section 真空计算

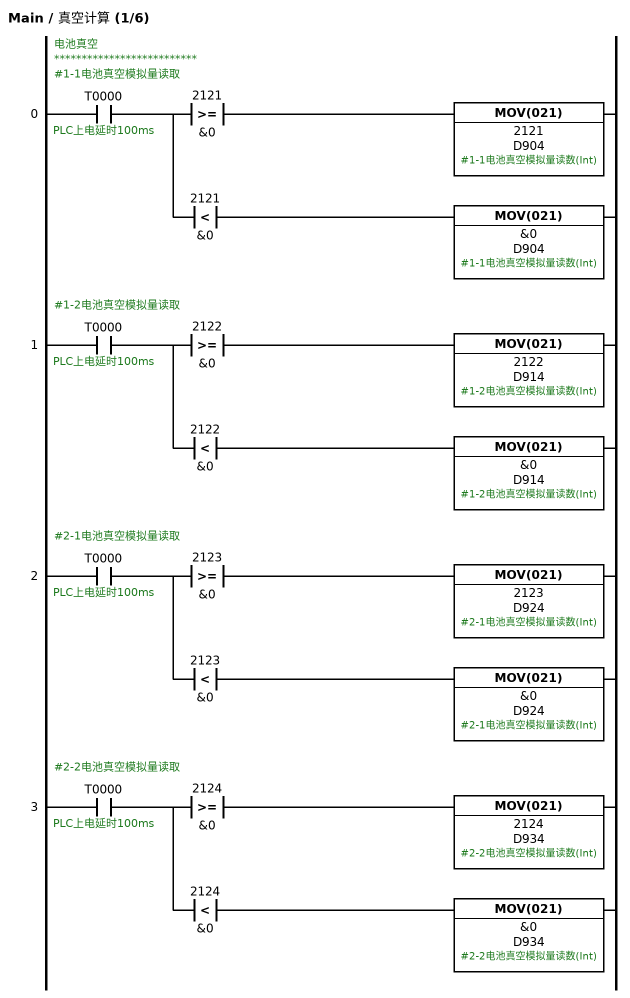
; rung 0: 电池真空 / ************************** / #1-1电池真空模拟量读取
LD T0000  ; PLC上电延时100ms
OUT TR0
AND>=S(327) 2121 &0
MOV(021) 2121 D904  ; #1-1电池真空模拟量读数(Int)
LD TR0
AND<S(312) 2121 &0
MOV(021) &0 D904  ; #1-1电池真空模拟量读数(Int)
; rung 1: #1-2电池真空模拟量读取
LD T0000  ; PLC上电延时100ms
OUT TR0
AND>=S(327) 2122 &0
MOV(021) 2122 D914  ; #1-2电池真空模拟量读数(Int)
LD TR0
AND<S(312) 2122 &0
MOV(021) &0 D914  ; #1-2电池真空模拟量读数(Int)
; rung 2: #2-1电池真空模拟量读取
LD T0000  ; PLC上电延时100ms
OUT TR0
AND>=S(327) 2123 &0
MOV(021) 2123 D924  ; #2-1电池真空模拟量读数(Int)
LD TR0
AND<S(312) 2123 &0
MOV(021) &0 D924  ; #2-1电池真空模拟量读数(Int)
; rung 3: #2-2电池真空模拟量读取
LD T0000  ; PLC上电延时100ms
OUT TR0
AND>=S(327) 2124 &0
MOV(021) 2124 D934  ; #2-2电池真空模拟量读数(Int)
LD TR0
AND<S(312) 2124 &0
MOV(021) &0 D934  ; #2-2电池真空模拟量读数(Int)

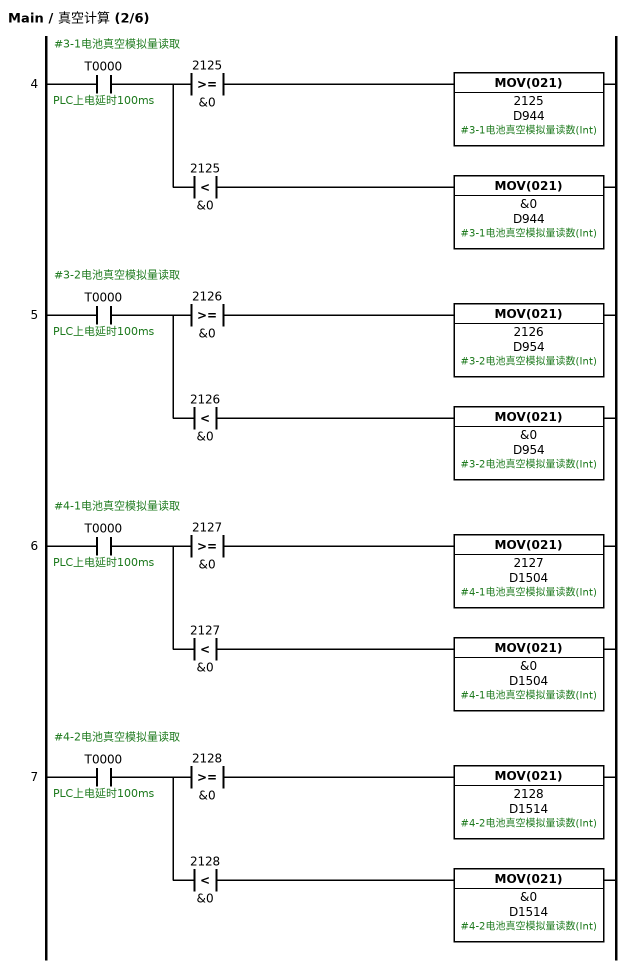
; rung 4: #3-1电池真空模拟量读取
LD T0000  ; PLC上电延时100ms
OUT TR0
AND>=S(327) 2125 &0
MOV(021) 2125 D944  ; #3-1电池真空模拟量读数(Int)
LD TR0
AND<S(312) 2125 &0
MOV(021) &0 D944  ; #3-1电池真空模拟量读数(Int)
; rung 5: #3-2电池真空模拟量读取
LD T0000  ; PLC上电延时100ms
OUT TR0
AND>=S(327) 2126 &0
MOV(021) 2126 D954  ; #3-2电池真空模拟量读数(Int)
LD TR0
AND<S(312) 2126 &0
MOV(021) &0 D954  ; #3-2电池真空模拟量读数(Int)
; rung 6: #4-1电池真空模拟量读取
LD T0000  ; PLC上电延时100ms
OUT TR0
AND>=S(327) 2127 &0
MOV(021) 2127 D1504  ; #4-1电池真空模拟量读数(Int)
LD TR0
AND<S(312) 2127 &0
MOV(021) &0 D1504  ; #4-1电池真空模拟量读数(Int)
; rung 7: #4-2电池真空模拟量读取
LD T0000  ; PLC上电延时100ms
OUT TR0
AND>=S(327) 2128 &0
MOV(021) 2128 D1514  ; #4-2电池真空模拟量读数(Int)
LD TR0
AND<S(312) 2128 &0
MOV(021) &0 D1514  ; #4-2电池真空模拟量读数(Int)

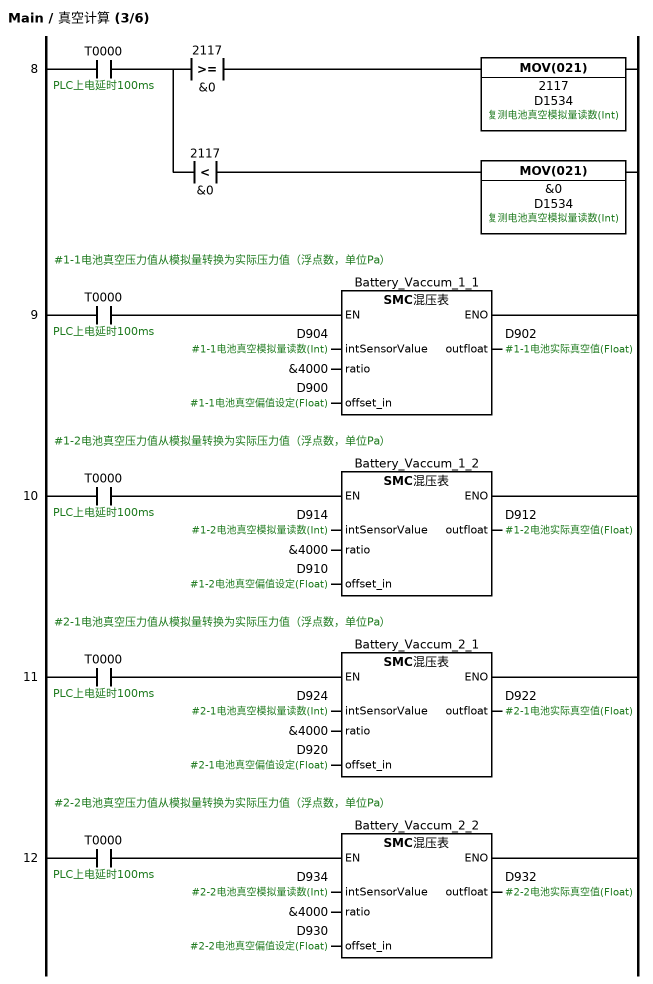
; rung 8
LD T0000  ; PLC上电延时100ms
OUT TR0
AND>=S(327) 2117 &0
MOV(021) 2117 D1534  ; 复测电池真空模拟量读数(Int)
LD TR0
AND<S(312) 2117 &0
MOV(021) &0 D1534  ; 复测电池真空模拟量读数(Int)
; rung 9: #1-1电池真空压力值从模拟量转换为实际压力值（浮点数，单位Pa）
LD T0000  ; PLC上电延时100ms
CALL Battery_Vaccum_1_1 : SMC混压表 (intSensorValue := D904, ratio := &4000, offset_in := D900, outfloat => D902)  ; #1-1电池真空模拟量读数(Int), #1-1电池真空偏值设定(Float), #1-1电池实际真空值(Float)
; rung 10: #1-2电池真空压力值从模拟量转换为实际压力值（浮点数，单位Pa）
LD T0000  ; PLC上电延时100ms
CALL Battery_Vaccum_1_2 : SMC混压表 (intSensorValue := D914, ratio := &4000, offset_in := D910, outfloat => D912)  ; #1-2电池真空模拟量读数(Int), #1-2电池真空偏值设定(Float), #1-2电池实际真空值(Float)
; rung 11: #2-1电池真空压力值从模拟量转换为实际压力值（浮点数，单位Pa）
LD T0000  ; PLC上电延时100ms
CALL Battery_Vaccum_2_1 : SMC混压表 (intSensorValue := D924, ratio := &4000, offset_in := D920, outfloat => D922)  ; #2-1电池真空模拟量读数(Int), #2-1电池真空偏值设定(Float), #2-1电池实际真空值(Float)
; rung 12: #2-2电池真空压力值从模拟量转换为实际压力值（浮点数，单位Pa）
LD T0000  ; PLC上电延时100ms
CALL Battery_Vaccum_2_2 : SMC混压表 (intSensorValue := D934, ratio := &4000, offset_in := D930, outfloat => D932)  ; #2-2电池真空模拟量读数(Int), #2-2电池真空偏值设定(Float), #2-2电池实际真空值(Float)

